C09095=1097.817,317.270,-83.466,178.547,18.904,152.358
C09096=1097.823,317.519,-83.498,178.550,18.907,152.358
C09097=1097.828,317.767,-83.529,178.553,18.909,152.358
C09098=1097.834,318.015,-83.561,178.556,18.912,152.358
C09099=1097.840,318.263,-83.593,178.560,18.915,152.358
C09100=1097.846,318.511,-83.625,178.563,18.918,152.358
C09101=1097.851,318.758,-83.657,178.566,18.920,152.359
C09102=1097.856,319.007,-83.689,178.569,18.923,152.359
C09103=1097.862,319.254,-83.721,178.572,18.926,152.359
C09104=1097.868,319.503,-83.753,178.575,18.928,152.359
C09105=1097.873,319.750,-83.785,178.578,18.931,152.359
C09106=1097.879,319.998,-83.817,178.583,18.934,152.359
C09107=1097.884,320.246,-83.848,178.586,18.937,152.359
C09108=1097.890,320.494,-83.880,178.589,18.939,152.359
C09109=1097.896,320.741,-83.912,178.592,18.942,152.359
C09110=1097.902,320.990,-83.944,178.595,18.945,152.359
C09111=1097.906,321.238,-83.976,178.598,18.948,152.359
C09112=1097.912,321.486,-84.008,178.601,18.951,152.359
C09113=1097.918,321.733,-84.040,178.604,18.954,152.359
C09114=1097.924,321.981,-84.072,178.607,18.956,152.359
C09115=1097.930,322.229,-84.105,178.611,18.959,152.359
C09116=1097.935,322.477,-84.136,178.614,18.961,152.360
C09117=1097.941,322.725,-84.169,178.618,18.965,152.360
C09118=1097.946,322.973,-84.201,178.621,18.967,152.360
C09119=1097.952,323.221,-84.233,178.624,18.970,152.360
C09120=1097.958,323.468,-84.266,178.627,18.973,152.360
C09121=1097.964,323.716,-84.297,178.630,18.975,152.360
C09122=1097.970,323.964,-84.329,178.633,18.979,152.360
C09123=1097.975,324.213,-84.362,178.637,18.981,152.360
C09124=1097.981,324.460,-84.394,178.640,18.984,152.360
C09125=1097.987,324.708,-84.426,178.643,18.987,152.360
C09126=1097.993,324.956,-84.458,178.646,18.990,152.360
C09127=1097.998,325.203,-84.491,178.649,18.993,152.360
C09128=1098.004,325.451,-84.523,178.652,18.996,152.361
C09129=1098.010,325.700,-84.555,178.655,18.998,152.361
C09130=1098.015,325.947,-84.588,178.658,19.001,152.361
C09131=1098.021,326.195,-84.620,178.661,19.004,152.361
C09132=1098.027,326.443,-84.652,178.665,19.007,152.361
C09133=1098.032,326.690,-84.685,178.668,19.010,152.361
C09134=1098.038,326.938,-84.717,178.671,19.013,152.361
C09135=1098.044,327.186,-84.750,178.674,19.016,152.361
C09136=1098.050,327.434,-84.782,178.678,19.019,152.361
C09137=1098.055,327.681,-84.814,178.681,19.022,152.362
C09138=1098.061,327.930,-84.847,178.684,19.024,152.362
C09139=1098.067,328.177,-84.880,178.687,19.027,152.362
C09140=1098.073,328.426,-84.912,178.691,19.030,152.362
C09141=1098.078,328.673,-84.945,178.694,19.033,152.362
C09142=1098.084,328.921,-84.977,178.697,19.036,152.362
C09143=1098.090,329.169,-85.010,178.700,19.039,152.362
C09144=1098.099,329.550,-85.060,178.705,19.044,152.362
C09145=1098.108,329.930,-85.109,178.710,19.047,152.362
C09146=1098.116,330.311,-85.160,178.715,19.052,152.363
C09147=1098.126,330.692,-85.210,178.720,19.057,152.363
C09148=1098.132,330.940,-85.242,178.723,19.060,152.363
C09149=1098.137,331.188,-85.276,178.726,19.063,152.363
C09150=1098.144,331.435,-85.309,178.729,19.066,152.363
C09151=1098.148,331.683,-85.341,178.733,19.069,152.363
C09152=1098.155,331.931,-85.374,178.735,19.072,152.364
C09153=1098.160,332.179,-85.407,178.738,19.075,152.364
C09154=1098.166,332.427,-85.439,178.742,19.078,152.364
C09155=1098.172,332.675,-85.472,178.745,19.081,152.364
C09156=1098.178,332.922,-85.505,178.748,19.084,152.364
C09157=1098.183,333.170,-85.538,178.751,19.087,152.364
C09158=1098.188,333.418,-85.571,178.755,19.090,152.364
C09159=1098.194,333.666,-85.603,178.757,19.094,152.365
C09160=1098.200,333.914,-85.637,178.760,19.096,152.365
C09161=1098.206,334.162,-85.670,178.764,19.100,152.365
C09162=1098.212,334.409,-85.703,178.767,19.103,152.365
C09163=1098.217,334.656,-85.736,178.770,19.106,152.365
C09164=1098.223,334.904,-85.768,178.773,19.110,152.366
C09165=1098.229,335.152,-85.802,178.776,19.112,152.366
C09166=1098.234,335.400,-85.835,178.779,19.115,152.366
C09167=1098.240,335.648,-85.868,178.783,19.119,152.366
C09168=1098.246,335.895,-85.901,178.786,19.122,152.366
C09169=1098.252,336.143,-85.935,178.789,19.125,152.367
C09170=1098.257,336.391,-85.968,178.792,19.129,152.367
C09171=1098.263,336.639,-86.001,178.795,19.131,152.367
C09172=1098.269,336.887,-86.034,178.798,19.135,152.367
C09173=1098.274,337.134,-86.067,178.802,19.138,152.367
C09174=1098.280,337.382,-86.100,178.805,19.141,152.367
C09175=1098.286,337.629,-86.133,178.808,19.145,152.368
C09176=1098.291,337.877,-86.166,178.811,19.148,152.368
C09177=1098.297,338.125,-86.200,178.814,19.151,152.368
C09178=1098.303,338.373,-86.232,178.818,19.154,152.368
C09179=1098.309,338.621,-86.266,178.820,19.157,152.368
C09180=1098.314,338.868,-86.299,178.823,19.161,152.369
C09181=1098.320,339.116,-86.333,178.827,19.164,152.369
C09182=1098.326,339.364,-86.366,178.830,19.167,152.369
C09183=1098.331,339.612,-86.400,178.833,19.171,152.369
C09184=1098.337,339.859,-86.433,178.836,19.174,152.370
C09185=1098.342,340.107,-86.467,178.839,19.177,152.370
C09186=1098.349,340.354,-86.500,178.842,19.181,152.370
C09187=1098.355,340.602,-86.533,178.845,19.184,152.370
C09188=1098.360,340.850,-86.567,178.849,19.188,152.371
C09189=1098.366,341.098,-86.600,178.851,19.191,152.371
C09190=1098.372,341.345,-86.634,178.854,19.194,152.371
C09191=1098.377,341.593,-86.667,178.858,19.198,152.371
C09192=1098.383,341.841,-86.701,178.861,19.201,152.372
C09193=1098.389,342.088,-86.735,178.864,19.205,152.372
C09194=1098.394,342.336,-86.768,178.867,19.208,152.372
C09195=1098.400,342.584,-86.802,178.870,19.211,152.372
C09196=1098.409,342.959,-86.852,178.875,19.216,152.373
C09197=1098.417,343.333,-86.903,178.880,19.222,152.373
C09198=1098.426,343.709,-86.955,178.885,19.227,152.373
C09199=1098.434,344.082,-87.006,178.889,19.232,152.374
C09200=1098.440,344.330,-87.039,178.892,19.236,152.374
C09201=1098.446,344.578,-87.074,178.895,19.239,152.374
C09202=1098.452,344.826,-87.107,178.899,19.243,152.375
C09203=1098.458,345.073,-87.141,178.901,19.246,152.375
C09204=1098.463,345.321,-87.174,178.905,19.250,152.375
C09205=1098.469,345.569,-87.208,178.908,19.253,152.376
C09206=1098.475,345.816,-87.242,178.911,19.257,152.376
C09207=1098.481,346.064,-87.276,178.914,19.260,152.376
C09208=1098.486,346.311,-87.310,178.916,19.263,152.376
C09209=1098.491,346.559,-87.344,178.920,19.267,152.377
C09210=1098.497,346.807,-87.378,178.923,19.271,152.377
C09211=1098.503,347.055,-87.412,178.926,19.274,152.377
C09212=1098.509,347.302,-87.446,178.929,19.278,152.378
C09213=1098.515,347.550,-87.480,178.932,19.282,152.378
C09214=1098.520,347.797,-87.514,178.935,19.285,152.378
C09215=1098.526,348.045,-87.548,178.939,19.289,152.379
C09216=1098.532,348.292,-87.582,178.941,19.292,152.379
C09217=1098.537,348.540,-87.616,178.945,19.296,152.379
C09218=1098.544,348.788,-87.650,178.947,19.300,152.380
C09219=1098.549,349.036,-87.684,178.951,19.303,152.380
C09220=1098.555,349.283,-87.718,178.953,19.307,152.380
C09221=1098.560,349.531,-87.752,178.957,19.311,152.380
C09222=1098.566,349.778,-87.787,178.960,19.315,152.381
C09223=1098.571,350.025,-87.821,178.963,19.318,152.381
C09224=1098.578,350.273,-87.855,178.966,19.322,152.381
C09225=1098.583,350.521,-87.889,178.969,19.326,152.382
C09226=1098.589,350.769,-87.923,178.972,19.330,152.382
C09227=1098.594,351.016,-87.957,178.975,19.333,152.383
C09228=1098.600,351.263,-87.991,178.979,19.337,152.383
C09229=1098.606,351.512,-88.027,178.981,19.340,152.383
C09230=1098.612,351.759,-88.061,178.985,19.344,152.384
C09231=1098.618,352.006,-88.095,178.987,19.348,152.384
C09232=1098.623,352.254,-88.129,178.991,19.352,152.384
C09233=1098.629,352.502,-88.164,178.993,19.355,152.385
C09234=1098.635,352.749,-88.198,178.997,19.359,152.385
C09235=1098.640,352.997,-88.232,179.000,19.363,152.385
C09236=1098.647,353.245,-88.267,179.003,19.367,152.386
C09237=1098.652,353.492,-88.301,179.006,19.371,152.386
C09238=1098.658,353.739,-88.336,179.009,19.374,152.387
C09239=1098.663,353.987,-88.371,179.012,19.379,152.387
C09240=1098.670,354.235,-88.405,179.014,19.382,152.387
C09241=1098.675,354.482,-88.440,179.018,19.386,152.388
C09242=1098.681,354.729,-88.474,179.021,19.390,152.388
C09243=1098.686,354.977,-88.509,179.024,19.394,152.388
C09244=1098.692,355.225,-88.543,179.027,19.398,152.389
C09245=1098.698,355.472,-88.578,179.030,19.402,152.389
C09246=1098.703,355.719,-88.612,179.033,19.406,152.390
C09247=1098.709,355.968,-88.647,179.036,19.410,152.390
C09248=1098.717,356.344,-88.700,179.041,19.416,152.391
C09249=1098.726,356.721,-88.753,179.045,19.422,152.391
C09250=1098.735,357.098,-88.806,179.050,19.428,152.392
C09251=1098.744,357.476,-88.859,179.055,19.434,152.393
C09252=1098.750,357.723,-88.894,179.057,19.438,152.393
C09253=1098.756,357.970,-88.929,179.060,19.442,152.393
C09254=1098.761,358.218,-88.964,179.064,19.446,152.394
C09255=1098.767,358.465,-88.998,179.066,19.450,152.394
C09256=1098.773,358.712,-89.033,179.069,19.454,152.395
C09257=1098.778,358.961,-89.068,179.073,19.458,152.395
C09258=1098.785,359.207,-89.103,179.075,19.462,152.396
C09259=1098.790,359.456,-89.138,179.079,19.466,152.396
C09260=1098.796,359.703,-89.173,179.082,19.471,152.397
C09261=1098.802,359.950,-89.207,179.084,19.475,152.397
C09262=1098.808,360.198,-89.243,179.088,19.479,152.397
C09263=1098.813,360.445,-89.278,179.091,19.483,152.398
C09264=1098.820,360.693,-89.313,179.093,19.487,152.398
C09265=1098.825,360.940,-89.347,179.096,19.491,152.399
C09266=1098.830,361.187,-89.383,179.100,19.495,152.399
C09267=1098.836,361.435,-89.418,179.102,19.499,152.400
C09268=1098.841,361.682,-89.453,179.105,19.504,152.400
C09269=1098.848,361.930,-89.488,179.109,19.508,152.401
C09270=1098.853,362.177,-89.524,179.111,19.512,152.401
C09271=1098.859,362.425,-89.559,179.114,19.517,152.402
C09272=1098.865,362.672,-89.594,179.117,19.521,152.402
C09273=1098.871,362.919,-89.629,179.120,19.525,152.403
C09274=1098.876,363.167,-89.664,179.123,19.529,152.403
C09275=1098.882,363.414,-89.699,179.126,19.534,152.404
C09276=1098.888,363.662,-89.735,179.129,19.538,152.404
C09277=1098.893,363.909,-89.770,179.132,19.542,152.405
C09278=1098.899,364.157,-89.805,179.135,19.546,152.405
C09279=1098.905,364.404,-89.841,179.138,19.551,152.406
C09280=1098.911,364.651,-89.876,179.140,19.555,152.406
C09281=1098.917,364.898,-89.911,179.144,19.559,152.407
C09282=1098.923,365.146,-89.947,179.147,19.563,152.407
C09283=1098.928,365.393,-89.982,179.150,19.568,152.408
C09284=1098.934,365.640,-90.018,179.152,19.572,152.408
C09285=1098.939,365.888,-90.053,179.156,19.576,152.409
C09286=1098.945,366.136,-90.088,179.159,19.581,152.410
C09287=1098.951,366.383,-90.124,179.162,19.586,152.410
C09288=1098.957,366.630,-90.159,179.164,19.590,152.411
C09289=1098.962,366.877,-90.195,179.167,19.594,152.411
C09290=1098.968,367.125,-90.230,179.170,19.599,152.412
C09291=1098.974,367.372,-90.266,179.173,19.604,152.412
C09292=1098.980,367.620,-90.302,179.175,19.608,152.413
C09293=1098.985,367.867,-90.337,179.179,19.612,152.414
C09294=1098.991,368.114,-90.373,179.182,19.617,152.414
C09295=1098.997,368.362,-90.408,179.185,19.621,152.415
C09296=1099.002,368.609,-90.444,179.188,19.626,152.415
C09297=1099.008,368.856,-90.481,179.190,19.630,152.416
C09298=1099.014,369.103,-90.516,179.193,19.635,152.416
C09299=1099.020,369.351,-90.552,179.196,19.640,152.417
C09300=1099.028,369.743,-90.608,179.201,19.647,152.418
C09301=1099.038,370.134,-90.665,179.205,19.654,152.419
C09302=1099.047,370.527,-90.722,179.210,19.662,152.420
C09303=1099.056,370.919,-90.778,179.214,19.669,152.421
C09304=1099.062,371.166,-90.815,179.217,19.674,152.422
C09305=1099.068,371.413,-90.850,179.220,19.678,152.422
C09306=1099.073,371.661,-90.886,179.223,19.683,152.423
C09307=1099.079,371.909,-90.922,179.226,19.688,152.423
C09308=1099.085,372.155,-90.958,179.229,19.693,152.424
C09309=1099.091,372.403,-90.994,179.231,19.697,152.425
C09310=1099.097,372.650,-91.030,179.234,19.702,152.425
C09311=1099.102,372.897,-91.066,179.237,19.706,152.426
C09312=1099.108,373.145,-91.102,179.240,19.711,152.427
C09313=1099.114,373.392,-91.138,179.243,19.716,152.427
C09314=1099.120,373.640,-91.174,179.246,19.721,152.428
C09315=1099.126,373.886,-91.210,179.249,19.726,152.429
C09316=1099.131,374.134,-91.247,179.251,19.730,152.429
C09317=1099.138,374.381,-91.283,179.254,19.735,152.430
C09318=1099.143,374.628,-91.318,179.257,19.740,152.431
C09319=1099.149,374.876,-91.355,179.260,19.745,152.431
C09320=1099.155,375.123,-91.391,179.263,19.750,152.432
C09321=1099.160,375.370,-91.428,179.266,19.755,152.433
C09322=1099.166,375.618,-91.464,179.269,19.760,152.433
C09323=1099.172,375.865,-91.500,179.272,19.765,152.434
C09324=1099.177,376.112,-91.536,179.275,19.770,152.435
C09325=1099.183,376.359,-91.572,179.277,19.775,152.436
C09326=1099.189,376.606,-91.609,179.280,19.779,152.436
C09327=1099.195,376.854,-91.645,179.283,19.784,152.437
C09328=1099.200,377.101,-91.682,179.286,19.789,152.438
C09329=1099.206,377.348,-91.718,179.288,19.795,152.439
C09330=1099.212,377.595,-91.754,179.291,19.800,152.439
C09331=1099.218,377.843,-91.791,179.294,19.805,152.440
C09332=1099.223,378.089,-91.827,179.297,19.810,152.441
C09333=1099.229,378.336,-91.864,179.300,19.815,152.441
C09334=1099.235,378.584,-91.900,179.302,19.820,152.442
C09335=1099.241,378.831,-91.937,179.305,19.825,152.443
C09336=1099.246,379.078,-91.973,179.308,19.831,152.444
C09337=1099.252,379.325,-92.010,179.311,19.835,152.444
C09338=1099.258,379.572,-92.047,179.314,19.841,152.445
C09339=1099.264,379.820,-92.083,179.317,19.846,152.446
C09340=1099.269,380.068,-92.120,179.319,19.851,152.447
C09341=1099.275,380.314,-92.156,179.322,19.856,152.448
C09342=1099.281,380.561,-92.193,179.325,19.861,152.448
C09343=1099.287,380.808,-92.229,179.328,19.867,152.449
C09344=1099.292,381.056,-92.267,179.331,19.872,152.450
C09345=1099.299,381.303,-92.303,179.333,19.877,152.451
C09346=1099.304,381.550,-92.340,179.336,19.882,152.452
C09347=1099.311,381.797,-92.376,179.339,19.887,152.452
C09348=1099.316,382.044,-92.413,179.342,19.893,152.453
C09349=1099.321,382.291,-92.450,179.344,19.898,152.454
C09350=1099.328,382.538,-92.487,179.347,19.903,152.455
C09351=1099.333,382.786,-92.524,179.350,19.909,152.456
C09352=1099.339,382.995,-92.555,179.352,19.913,152.456
C09353=1099.343,383.204,-92.586,179.354,19.917,152.457
C09354=1099.348,383.415,-92.617,179.356,19.922,152.458
C09355=1099.353,383.624,-92.649,179.359,19.927,152.458
C09356=1099.358,383.834,-92.680,179.361,19.931,152.459
C09357=1099.363,384.042,-92.712,179.363,19.936,152.460
C09358=1099.368,384.252,-92.743,179.366,19.941,152.461
C09359=1099.372,384.463,-92.774,179.368,19.946,152.461
C09360=1099.378,384.709,-92.811,179.371,19.951,152.462
C09361=1099.384,384.956,-92.848,179.374,19.956,152.463
C09362=1099.389,385.203,-92.885,179.376,19.962,152.464
C09363=1099.395,385.451,-92.922,179.379,19.967,152.465
C09364=1099.401,385.697,-92.960,179.381,19.973,152.466
C09365=1099.407,385.945,-92.997,179.384,19.978,152.467
C09366=1099.413,386.192,-93.034,179.387,19.984,152.467
C09367=1099.419,386.439,-93.071,179.390,19.990,152.468
C09368=1099.424,386.686,-93.108,179.393,19.995,152.469
C09369=1099.430,386.933,-93.145,179.395,20.001,152.470
C09370=1099.436,387.180,-93.183,179.398,20.007,152.471
C09371=1099.441,387.427,-93.220,179.400,20.012,152.472
C09372=1099.447,387.675,-93.257,179.403,20.018,152.473
C09373=1099.454,387.921,-93.294,179.406,20.023,152.474
C09374=1099.459,388.169,-93.331,179.408,20.029,152.475
C09375=1099.465,388.415,-93.369,179.412,20.035,152.476
C09376=1099.471,388.663,-93.406,179.414,20.041,152.477
C09377=1099.477,388.909,-93.444,179.417,20.047,152.478
C09378=1099.482,389.157,-93.481,179.419,20.052,152.479
C09379=1099.488,389.403,-93.519,179.422,20.058,152.479
C09380=1099.494,389.651,-93.556,179.425,20.063,152.480
C09381=1099.500,389.898,-93.594,179.428,20.070,152.481
C09382=1099.506,390.144,-93.631,179.430,20.075,152.482
C09383=1099.511,390.392,-93.668,179.433,20.081,152.483
C09384=1099.517,390.638,-93.706,179.435,20.087,152.484
C09385=1099.523,390.886,-93.743,179.438,20.093,152.485
C09386=1099.529,391.133,-93.781,179.440,20.098,152.486
C09387=1099.535,391.379,-93.819,179.444,20.105,152.487
C09388=1099.540,391.627,-93.856,179.446,20.110,152.488
C09389=1099.546,391.873,-93.894,179.449,20.116,152.489
C09390=1099.553,392.121,-93.932,179.451,20.122,152.490
C09391=1099.558,392.368,-93.969,179.454,20.128,152.491
C09392=1099.564,392.615,-94.006,179.457,20.134,152.492
C09393=1099.570,392.862,-94.044,179.459,20.141,152.493
C09394=1099.576,393.108,-94.082,179.462,20.146,152.494
C09395=1099.582,393.355,-94.120,179.464,20.152,152.495
C09396=1099.587,393.603,-94.157,179.467,20.159,152.496
C09397=1099.593,393.850,-94.195,179.470,20.165,152.498
C09398=1099.599,394.097,-94.233,179.472,20.171,152.499
C09399=1099.605,394.344,-94.271,179.475,20.177,152.500
C09400=1099.611,394.591,-94.309,179.478,20.184,152.501
C09401=1099.616,394.838,-94.347,179.480,20.189,152.502
C09402=1099.622,395.084,-94.385,179.482,20.195,152.503
C09403=1099.628,395.332,-94.423,179.485,20.202,152.504
C09404=1099.634,395.579,-94.461,179.488,20.208,152.505
C09405=1099.639,395.826,-94.499,179.490,20.214,152.506
C09406=1099.645,396.072,-94.537,179.493,20.221,152.507
C09407=1099.651,396.319,-94.575,179.495,20.227,152.508
C09408=1099.656,396.536,-94.607,179.497,20.233,152.509
C09409=1099.661,396.752,-94.641,179.500,20.238,152.510
C09410=1099.666,396.967,-94.674,179.502,20.243,152.511
C09411=1099.672,397.183,-94.707,179.504,20.249,152.512
C09412=1099.677,397.399,-94.741,179.507,20.255,152.513
C09413=1099.681,397.615,-94.775,179.508,20.260,152.514
C09414=1099.687,397.831,-94.808,179.511,20.266,152.515
C09415=1099.691,398.046,-94.841,179.513,20.272,152.516
C09416=1099.698,398.294,-94.879,179.516,20.278,152.518
C09417=1099.703,398.541,-94.917,179.518,20.284,152.519
C09418=1099.709,398.787,-94.956,179.521,20.291,152.520
C09419=1099.715,399.035,-94.994,179.523,20.298,152.521
C09420=1099.721,399.281,-95.032,179.525,20.304,152.522
C09421=1099.727,399.528,-95.070,179.528,20.311,152.523
C09422=1099.733,399.776,-95.109,179.531,20.317,152.525
C09423=1099.739,400.022,-95.147,179.533,20.323,152.526
C09424=1099.744,400.269,-95.185,179.536,20.331,152.527
C09425=1099.750,400.517,-95.224,179.538,20.337,152.528
C09426=1099.756,400.763,-95.263,179.541,20.344,152.529
C09427=1099.761,401.010,-95.301,179.543,20.350,152.531
C09428=1099.768,401.257,-95.339,179.545,20.357,152.532
C09429=1099.773,401.504,-95.378,179.548,20.364,152.533
C09430=1099.779,401.751,-95.416,179.550,20.371,152.534
C09431=1099.785,401.998,-95.455,179.553,20.378,152.536
C09432=1099.790,402.245,-95.494,179.555,20.384,152.537
C09433=1099.797,402.492,-95.532,179.558,20.391,152.538
C09434=1099.802,402.739,-95.571,179.560,20.398,152.539
C09435=1099.808,402.985,-95.609,179.563,20.405,152.541
C09436=1099.814,403.233,-95.648,179.565,20.412,152.542
C09437=1099.819,403.480,-95.686,179.568,20.418,152.543
C09438=1099.826,403.726,-95.725,179.570,20.426,152.545
C09439=1099.831,403.973,-95.764,179.572,20.432,152.546
C09440=1099.837,404.221,-95.803,179.575,20.439,152.547
C09441=1099.843,404.467,-95.841,179.577,20.446,152.549
C09442=1099.849,404.714,-95.880,179.580,20.453,152.550
C09443=1099.855,404.961,-95.919,179.583,20.461,152.551
C09444=1099.861,405.208,-95.957,179.585,20.467,152.552
C09445=1099.867,405.455,-95.997,179.588,20.475,152.554
C09446=1099.872,405.701,-96.036,179.590,20.482,152.555
C09447=1099.878,405.949,-96.074,179.593,20.489,152.557
C09448=1099.884,406.195,-96.113,179.595,20.496,152.558
C09449=1099.890,406.442,-96.152,179.597,20.504,152.559
C09450=1099.896,406.689,-96.191,179.599,20.510,152.561
C09451=1099.902,406.936,-96.230,179.602,20.518,152.562
C09452=1099.907,407.183,-96.269,179.605,20.525,152.564
C09453=1099.913,407.430,-96.308,179.607,20.532,152.565
C09454=1099.919,407.676,-96.348,179.609,20.540,152.566
C09455=1099.925,407.924,-96.386,179.611,20.547,152.568
C09456=1099.931,408.170,-96.425,179.614,20.554,152.569
C09457=1099.937,408.417,-96.464,179.617,20.562,152.571
C09458=1099.942,408.664,-96.503,179.619,20.569,152.572
C09459=1099.948,408.911,-96.543,179.621,20.577,152.573
C09460=1099.954,409.157,-96.582,179.624,20.584,152.575
C09461=1099.960,409.405,-96.621,179.626,20.592,152.576
C09462=1099.966,409.652,-96.661,179.629,20.599,152.578
C09463=1099.971,409.898,-96.700,179.631,20.607,152.579
C09464=1099.976,410.114,-96.734,179.633,20.614,152.581
C09465=1099.981,410.331,-96.768,179.635,20.621,152.582
C09466=1099.986,410.546,-96.803,179.637,20.627,152.583
C09467=1099.992,410.763,-96.837,179.640,20.634,152.584
C09468=1099.996,410.978,-96.872,179.642,20.641,152.586
C09469=1100.001,411.194,-96.906,179.644,20.647,152.587
C09470=1100.007,411.410,-96.941,179.646,20.654,152.589
C09471=1100.012,411.626,-96.975,179.648,20.661,152.590
C09472=1100.018,411.873,-97.015,179.650,20.668,152.591
C09473=1100.023,412.119,-97.054,179.652,20.676,152.593
C09474=1100.029,412.366,-97.094,179.655,20.684,152.594
C09475=1100.035,412.614,-97.133,179.657,20.692,152.596
C09476=1100.041,412.860,-97.172,179.660,20.699,152.597
C09477=1100.047,413.107,-97.212,179.661,20.707,152.599
C09478=1100.053,413.354,-97.252,179.664,20.715,152.601
C09479=1100.059,413.600,-97.291,179.667,20.723,152.602
C09480=1100.065,413.847,-97.330,179.669,20.731,152.604
C09481=1100.071,414.094,-97.371,179.671,20.739,152.605
C09482=1100.076,414.340,-97.410,179.674,20.747,152.607
C09483=1100.082,414.588,-97.450,179.676,20.755,152.609
C09484=1100.088,414.834,-97.490,179.678,20.763,152.610
C09485=1100.094,415.081,-97.529,179.681,20.771,152.612
C09486=1100.100,415.327,-97.569,179.683,20.779,152.613
C09487=1100.106,415.574,-97.608,179.686,20.787,152.615
C09488=1100.112,415.821,-97.649,179.688,20.796,152.617
C09489=1100.118,416.068,-97.689,179.690,20.804,152.618
C09490=1100.124,416.314,-97.728,179.693,20.812,152.620
C09491=1100.130,416.561,-97.768,179.694,20.820,152.622
C09492=1100.136,416.808,-97.808,179.697,20.828,152.623
C09493=1100.142,417.055,-97.848,179.699,20.837,152.625
C09494=1100.147,417.301,-97.888,179.701,20.845,152.627
C09495=1100.153,417.548,-97.928,179.704,20.853,152.628
C09496=1100.159,417.795,-97.968,179.706,20.862,152.630
C09497=1100.166,418.041,-98.008,179.708,20.870,152.632
C09498=1100.170,418.288,-98.048,179.711,20.879,152.634
C09499=1100.177,418.535,-98.088,179.713,20.887,152.635
C09500=1100.182,418.781,-98.129,179.715,20.896,152.637
C09501=1100.188,419.029,-98.168,179.718,20.904,152.639
C09502=1100.195,419.275,-98.208,179.720,20.913,152.641
C09503=1100.200,419.521,-98.249,179.722,20.922,152.643
C09504=1100.206,419.768,-98.289,179.724,20.930,152.644
C09505=1100.212,420.015,-98.329,179.727,20.939,152.646
C09506=1100.218,420.262,-98.369,179.729,20.947,152.648
C09507=1100.223,420.509,-98.410,179.731,20.956,152.650
C09508=1100.230,420.755,-98.450,179.733,20.965,152.651
C09509=1100.236,421.002,-98.491,179.735,20.973,152.653
C09510=1100.241,421.248,-98.530,179.738,20.982,152.655
C09511=1100.247,421.494,-98.571,179.740,20.992,152.657
C09512=1100.253,421.741,-98.611,179.743,21.000,152.659
C09513=1100.259,421.988,-98.652,179.745,21.009,152.661
C09514=1100.265,422.234,-98.692,179.747,21.018,152.663
C09515=1100.271,422.481,-98.733,179.749,21.027,152.664
C09516=1100.277,422.728,-98.773,179.751,21.036,152.666
C09517=1100.283,422.975,-98.814,179.753,21.045,152.668
C09518=1100.289,423.221,-98.854,179.755,21.054,152.670
C09519=1100.295,423.468,-98.895,179.758,21.064,152.672
C09520=1100.300,423.690,-98.931,179.760,21.071,152.674
C09521=1100.305,423.913,-98.968,179.762,21.080,152.675
C09522=1100.310,424.136,-99.004,179.764,21.088,152.677
C09523=1100.316,424.358,-99.042,179.766,21.096,152.679
C09524=1100.322,424.581,-99.078,179.767,21.104,152.681
C09525=1100.327,424.804,-99.115,179.770,21.113,152.683
C09526=1100.332,425.027,-99.152,179.772,21.122,152.684
C09527=1100.337,425.250,-99.188,179.773,21.130,152.686
C09528=1100.343,425.496,-99.229,179.775,21.139,152.688
C09529=1100.349,425.743,-99.270,179.778,21.149,152.690
C09530=1100.354,425.989,-99.311,179.780,21.158,152.692
C09531=1100.361,426.236,-99.351,179.782,21.167,152.694
C09532=1100.367,426.482,-99.393,179.784,21.177,152.696
C09533=1100.372,426.729,-99.433,179.787,21.187,152.698
C09534=1100.378,426.975,-99.475,179.789,21.196,152.700
C09535=1100.384,427.222,-99.516,179.791,21.205,152.702
C09536=1100.390,427.468,-99.556,179.793,21.215,152.704
C09537=1100.396,427.715,-99.597,179.795,21.225,152.706
C09538=1100.402,427.961,-99.638,179.797,21.234,152.709
C09539=1100.408,428.208,-99.679,179.799,21.244,152.711
C09540=1100.414,428.454,-99.721,179.802,21.254,152.713
C09541=1100.421,428.701,-99.761,179.804,21.264,152.715
C09542=1100.427,428.947,-99.803,179.805,21.273,152.717
C09543=1100.432,429.194,-99.844,179.808,21.283,152.719
C09544=1100.438,429.440,-99.885,179.810,21.293,152.721
C09545=1100.444,429.687,-99.927,179.812,21.304,152.724
C09546=1100.450,429.933,-99.967,179.814,21.313,152.726
C09547=1100.456,430.180,-100.009,179.816,21.323,152.728
C09548=1100.462,430.426,-100.050,179.818,21.334,152.730
C09549=1100.467,430.673,-100.091,179.820,21.343,152.732
C09550=1100.473,430.919,-100.132,179.823,21.354,152.734
C09551=1100.479,431.165,-100.174,179.824,21.364,152.737
C09552=1100.485,431.411,-100.215,179.826,21.374,152.739
C09553=1100.492,431.658,-100.257,179.829,21.384,152.741
C09554=1100.498,431.905,-100.298,179.830,21.394,152.743
C09555=1100.503,432.151,-100.339,179.833,21.405,152.746
C09556=1100.509,432.397,-100.381,179.834,21.415,152.748
C09557=1100.515,432.644,-100.422,179.837,21.426,152.750
C09558=1100.521,432.890,-100.464,179.838,21.436,152.753
C09559=1100.527,433.136,-100.506,179.841,21.446,152.755
C09560=1100.533,433.383,-100.548,179.843,21.457,152.757
C09561=1100.539,433.629,-100.589,179.845,21.467,152.759
C09562=1100.545,433.876,-100.631,179.846,21.478,152.762
C09563=1100.551,434.122,-100.672,179.849,21.488,152.764
C09564=1100.556,434.368,-100.714,179.850,21.499,152.767
C09565=1100.562,434.615,-100.755,179.853,21.510,152.769
C09566=1100.569,434.861,-100.797,179.854,21.520,152.771
C09567=1100.575,435.108,-100.839,179.856,21.532,152.774
C09568=1100.580,435.354,-100.882,179.858,21.542,152.776
C09569=1100.586,435.600,-100.923,179.860,21.553,152.779
C09570=1100.592,435.846,-100.964,179.862,21.564,152.781
C09571=1100.599,436.093,-101.006,179.864,21.575,152.784
C09572=1100.604,436.339,-101.048,179.866,21.586,152.786
C09573=1100.610,436.585,-101.090,179.868,21.596,152.788
C09574=1100.616,436.831,-101.132,179.870,21.608,152.791
C09575=1100.622,437.078,-101.174,179.872,21.619,152.794
C09576=1100.630,437.434,-101.235,179.874,21.635,152.797
C09577=1100.639,437.789,-101.296,179.877,21.651,152.801
C09578=1100.648,438.146,-101.356,179.879,21.667,152.804
C09579=1100.656,438.502,-101.418,179.882,21.684,152.808
C09580=1100.663,438.748,-101.460,179.884,21.695,152.811
C09581=1100.669,438.995,-101.502,179.886,21.706,152.813
C09582=1100.674,439.241,-101.544,179.888,21.718,152.816
C09583=1100.681,439.487,-101.586,179.890,21.730,152.819
C09584=1100.687,439.733,-101.628,179.892,21.741,152.821
C09585=1100.692,439.980,-101.670,179.893,21.752,152.824
C09586=1100.699,440.226,-101.713,179.895,21.764,152.826
C09587=1100.705,440.472,-101.756,179.897,21.776,152.829
C09588=1100.711,440.718,-101.797,179.899,21.788,152.832
C09589=1100.717,440.965,-101.840,179.900,21.799,152.835
C09590=1100.723,441.210,-101.882,179.902,21.811,152.837
C09591=1100.729,441.457,-101.925,179.904,21.823,152.840
C09592=1100.734,441.703,-101.968,179.906,21.835,152.843
C09593=1100.740,441.949,-102.010,179.907,21.846,152.845
C09594=1100.747,442.195,-102.053,179.909,21.858,152.848
C09595=1100.753,442.441,-102.095,179.911,21.871,152.851
C09596=1100.758,442.687,-102.138,179.913,21.883,152.854
C09597=1100.764,442.934,-102.180,179.915,21.895,152.857
C09598=1100.770,443.180,-102.222,179.917,21.907,152.859
C09599=1100.777,443.426,-102.266,179.918,21.919,152.862
C09600=1100.782,443.672,-102.308,179.919,21.931,152.865
C09601=1100.789,443.918,-102.351,179.921,21.944,152.868
C09602=1100.794,444.164,-102.394,179.922,21.956,152.871
C09603=1100.801,444.411,-102.437,179.924,21.968,152.874
C09604=1100.806,444.657,-102.480,179.925,21.980,152.877
C09605=1100.813,444.903,-102.522,179.926,21.992,152.880
C09606=1100.818,445.149,-102.565,179.926,22.005,152.883
C09607=1100.825,445.396,-102.608,179.927,22.017,152.886
C09608=1100.830,445.641,-102.651,179.927,22.028,152.889
C09609=1100.837,445.888,-102.693,179.928,22.041,152.892
C09610=1100.843,446.133,-102.737,179.928,22.053,152.895
C09611=1100.849,446.380,-102.780,179.928,22.065,152.898
C09612=1100.854,446.626,-102.823,179.928,22.077,152.901
C09613=1100.861,446.872,-102.866,179.928,22.089,152.904
C09614=1100.866,447.118,-102.909,179.928,22.101,152.907
C09615=1100.872,447.365,-102.952,179.927,22.113,152.910
C09616=1100.879,447.611,-102.996,179.926,22.125,152.913
C09617=1100.884,447.856,-103.038,179.925,22.137,152.916
C09618=1100.890,448.103,-103.081,179.925,22.149,152.920
C09619=1100.896,448.349,-103.124,179.924,22.161,152.923
C09620=1100.903,448.595,-103.167,179.923,22.173,152.926
C09621=1100.909,448.841,-103.211,179.923,22.185,152.929
C09622=1100.915,449.087,-103.253,179.921,22.197,152.932
C09623=1100.921,449.333,-103.297,179.919,22.209,152.936
C09624=1100.926,449.579,-103.340,179.918,22.221,152.939
C09625=1100.933,449.826,-103.383,179.917,22.233,152.942
C09626=1100.938,450.071,-103.427,179.915,22.244,152.945
C09627=1100.945,450.317,-103.470,179.914,22.256,152.948
C09628=1100.547,450.310,-103.615,179.847,22.478,153.015
C09629=1100.541,450.064,-103.571,179.849,22.467,153.012
C09630=1100.534,449.818,-103.529,179.850,22.454,153.008
C09631=1100.528,449.571,-103.485,179.851,22.442,153.005
C09632=1100.522,449.326,-103.442,179.853,22.431,153.002
C09633=1100.516,449.080,-103.399,179.854,22.419,152.999
C09634=1100.510,448.834,-103.355,179.855,22.407,152.996
C09635=1100.504,448.588,-103.312,179.856,22.395,152.992
C09636=1100.498,448.341,-103.269,179.857,22.383,152.989
C09637=1100.492,448.096,-103.226,179.858,22.370,152.986
C09638=1100.486,447.849,-103.182,179.859,22.359,152.983
C09639=1100.480,447.603,-103.139,179.859,22.346,152.980
C09640=1100.474,447.357,-103.096,179.860,22.334,152.976
C09641=1100.468,447.111,-103.053,179.860,22.322,152.973
C09642=1100.462,446.865,-103.010,179.860,22.310,152.970
C09643=1100.456,446.618,-102.967,179.860,22.298,152.967
C09644=1100.450,446.372,-102.923,179.860,22.286,152.964
C09645=1100.444,446.126,-102.880,179.861,22.274,152.961
C09646=1100.437,445.880,-102.838,179.860,22.261,152.958
C09647=1100.432,445.634,-102.795,179.860,22.249,152.955
C09648=1100.426,445.388,-102.752,179.859,22.237,152.952
C09649=1100.420,445.142,-102.709,179.858,22.225,152.949
C09650=1100.414,444.896,-102.665,179.857,22.212,152.946
C09651=1100.407,444.650,-102.623,179.856,22.200,152.943
C09652=1100.401,444.404,-102.580,179.855,22.188,152.940
C09653=1100.395,444.157,-102.537,179.855,22.176,152.937
C09654=1100.390,443.911,-102.494,179.853,22.163,152.934
C09655=1100.383,443.665,-102.451,179.852,22.151,152.931
C09656=1100.377,443.419,-102.409,179.850,22.139,152.928
C09657=1100.372,443.173,-102.366,179.848,22.127,152.926
C09658=1100.366,442.926,-102.323,179.846,22.114,152.923
C09659=1100.359,442.681,-102.281,179.844,22.102,152.920
C09660=1100.353,442.434,-102.237,179.842,22.090,152.917
C09661=1100.348,442.188,-102.195,179.841,22.078,152.914
C09662=1100.341,441.942,-102.152,179.839,22.066,152.911
C09663=1100.336,441.696,-102.110,179.837,22.054,152.909
C09664=1100.329,441.450,-102.068,179.835,22.041,152.906
C09665=1100.323,441.203,-102.025,179.833,22.029,152.903
C09666=1100.318,440.958,-101.982,179.832,22.018,152.900
C09667=1100.311,440.711,-101.939,179.830,22.006,152.898
C09668=1100.306,440.465,-101.897,179.828,21.994,152.895
C09669=1100.299,440.219,-101.855,179.826,21.982,152.892
C09670=1100.293,439.973,-101.812,179.824,21.971,152.890
C09671=1100.287,439.726,-101.771,179.822,21.959,152.887
C09672=1100.280,439.480,-101.728,179.820,21.948,152.884
C09673=1100.275,439.234,-101.685,179.818,21.936,152.882
C09674=1100.269,438.988,-101.644,179.817,21.925,152.879
C09675=1100.263,438.741,-101.601,179.814,21.913,152.877
C09676=1100.257,438.495,-101.559,179.812,21.902,152.874
C09677=1100.248,438.146,-101.499,179.810,21.886,152.870
C09678=1100.240,437.797,-101.439,179.807,21.870,152.867
C09679=1100.231,437.449,-101.380,179.804,21.854,152.863
C09680=1100.223,437.100,-101.321,179.802,21.838,152.860
C09681=1100.217,436.853,-101.278,179.800,21.827,152.857
C09682=1100.210,436.607,-101.236,179.797,21.815,152.854
C09683=1100.205,436.361,-101.195,179.796,21.804,152.852
C09684=1100.199,436.115,-101.152,179.794,21.793,152.850
C09685=1100.192,435.868,-101.110,179.791,21.782,152.847
C09686=1100.187,435.622,-101.068,179.790,21.771,152.845
C09687=1100.181,435.376,-101.026,179.788,21.760,152.842
C09688=1100.175,435.130,-100.985,179.786,21.750,152.840
C09689=1100.168,434.883,-100.942,179.784,21.739,152.837
C09690=1100.163,434.637,-100.900,179.782,21.728,152.835
C09691=1100.157,434.391,-100.859,179.780,21.717,152.833
C09692=1100.151,434.144,-100.817,179.778,21.706,152.830
C09693=1100.145,433.898,-100.776,179.776,21.696,152.828
C09694=1100.140,433.651,-100.734,179.773,21.685,152.825
C09695=1100.134,433.405,-100.692,179.772,21.674,152.823
C09696=1100.128,433.158,-100.651,179.769,21.663,152.821
C09697=1100.122,432.912,-100.609,179.768,21.653,152.818
C09698=1100.116,432.666,-100.568,179.766,21.643,152.816
C09699=1100.110,432.420,-100.526,179.763,21.632,152.814
C09700=1100.103,432.173,-100.484,179.762,21.622,152.811
C09701=1100.097,431.927,-100.443,179.759,21.612,152.809
C09702=1100.091,431.681,-100.402,179.758,21.601,152.807
C09703=1100.085,431.434,-100.360,179.755,21.591,152.805
C09704=1100.080,431.188,-100.318,179.753,21.581,152.802
C09705=1100.074,430.942,-100.277,179.751,21.570,152.800
C09706=1100.069,430.695,-100.236,179.749,21.560,152.798
C09707=1100.062,430.448,-100.194,179.747,21.550,152.796
C09708=1100.056,430.202,-100.153,179.744,21.540,152.794
C09709=1100.050,429.956,-100.111,179.743,21.530,152.791
C09710=1100.045,429.709,-100.070,179.740,21.520,152.789
C09711=1100.039,429.462,-100.029,179.738,21.510,152.787
C09712=1100.033,429.216,-99.987,179.737,21.500,152.785
C09713=1100.027,428.970,-99.946,179.734,21.489,152.783
C09714=1100.020,428.724,-99.906,179.732,21.480,152.780
C09715=1100.014,428.477,-99.864,179.730,21.470,152.778
C09716=1100.009,428.231,-99.824,179.727,21.460,152.776
C09717=1100.002,427.984,-99.782,179.725,21.451,152.774
C09718=1099.997,427.737,-99.741,179.723,21.441,152.772
C09719=1099.991,427.491,-99.700,179.721,21.431,152.770
C09720=1099.984,427.245,-99.659,179.719,21.421,152.768
C09721=1099.978,426.998,-99.618,179.717,21.412,152.766
C09722=1099.973,426.751,-99.577,179.715,21.402,152.764
C09723=1099.967,426.505,-99.536,179.712,21.392,152.762
C09724=1099.961,426.258,-99.495,179.710,21.383,152.760
C09725=1099.954,426.012,-99.454,179.708,21.374,152.758
C09726=1099.949,425.765,-99.413,179.706,21.364,152.756
C09727=1099.943,425.518,-99.373,179.703,21.355,152.754
C09728=1099.937,425.272,-99.331,179.701,21.345,152.752
C09729=1099.932,425.050,-99.295,179.699,21.336,152.750
C09730=1099.927,424.826,-99.257,179.698,21.328,152.748
C09731=1099.921,424.603,-99.221,179.695,21.320,152.746
C09732=1099.915,424.380,-99.184,179.694,21.311,152.744
C09733=1099.911,424.157,-99.147,179.691,21.303,152.743
C09734=1099.905,423.934,-99.111,179.689,21.294,152.741
C09735=1099.900,423.711,-99.073,179.688,21.286,152.739
C09736=1099.894,423.488,-99.037,179.685,21.277,152.737
C09737=1099.889,423.241,-98.996,179.683,21.268,152.735
C09738=1099.882,422.994,-98.956,179.681,21.259,152.733
C09739=1099.877,422.747,-98.915,179.679,21.251,152.732
C09740=1099.871,422.501,-98.874,179.677,21.241,152.730
C09741=1099.865,422.255,-98.835,179.674,21.232,152.728
C09742=1099.860,422.008,-98.794,179.671,21.223,152.726
C09743=1099.853,421.761,-98.754,179.669,21.214,152.724
C09744=1099.847,421.515,-98.712,179.667,21.205,152.722
C09745=1099.841,421.268,-98.673,179.665,21.196,152.720
C09746=1099.835,421.021,-98.632,179.663,21.188,152.718
C09747=1099.829,420.775,-98.592,179.660,21.179,152.717
C09748=1099.823,420.528,-98.551,179.658,21.170,152.715
C09749=1099.817,420.281,-98.511,179.656,21.161,152.713
C09750=1099.811,420.035,-98.470,179.654,21.152,152.711
C09751=1099.806,419.789,-98.430,179.651,21.144,152.709
C09752=1099.800,419.542,-98.390,179.649,21.135,152.707
C09753=1099.794,419.295,-98.350,179.647,21.126,152.706
C09754=1099.788,419.048,-98.310,179.645,21.118,152.704
C09755=1099.782,418.801,-98.269,179.642,21.109,152.702
C09756=1099.776,418.555,-98.229,179.640,21.101,152.700
C09757=1099.770,418.309,-98.189,179.638,21.092,152.699
C09758=1099.764,418.062,-98.149,179.635,21.083,152.697
C09759=1099.759,417.815,-98.109,179.633,21.075,152.695
C09760=1099.752,417.568,-98.069,179.631,21.066,152.693
C09761=1099.746,417.321,-98.029,179.628,21.058,152.692
C09762=1099.741,417.075,-97.989,179.626,21.049,152.690
C09763=1099.735,416.829,-97.949,179.623,21.041,152.688
C09764=1099.730,416.581,-97.909,179.621,21.033,152.687
C09765=1099.723,416.335,-97.868,179.619,21.024,152.685
C09766=1099.718,416.088,-97.829,179.616,21.016,152.683
C09767=1099.711,415.842,-97.789,179.614,21.007,152.681
C09768=1099.705,415.595,-97.750,179.611,21.000,152.680
C09769=1099.700,415.348,-97.709,179.609,20.992,152.678
C09770=1099.694,415.101,-97.670,179.607,20.984,152.677
C09771=1099.688,414.855,-97.630,179.605,20.975,152.675
C09772=1099.682,414.608,-97.590,179.602,20.967,152.673
C09773=1099.675,414.361,-97.550,179.599,20.959,152.672
C09774=1099.669,414.114,-97.511,179.597,20.951,152.670
C09775=1099.665,413.867,-97.471,179.595,20.942,152.668
C09776=1099.658,413.621,-97.431,179.593,20.935,152.667
C09777=1099.652,413.374,-97.392,179.590,20.927,152.665
C09778=1099.647,413.127,-97.353,179.588,20.919,152.664
C09779=1099.640,412.881,-97.312,179.585,20.911,152.662
C09780=1099.634,412.633,-97.273,179.583,20.903,152.661
C09781=1099.628,412.386,-97.234,179.581,20.895,152.659
C09782=1099.623,412.140,-97.194,179.578,20.888,152.658
C09783=1099.616,411.893,-97.154,179.576,20.880,152.656
C09784=1099.611,411.647,-97.115,179.573,20.872,152.654
C09785=1099.606,411.430,-97.080,179.571,20.865,152.653
C09786=1099.601,411.214,-97.045,179.569,20.858,152.652
C09787=1099.596,410.998,-97.011,179.567,20.851,152.650
C09788=1099.591,410.781,-96.977,179.565,20.844,152.649
C09789=1099.585,410.565,-96.942,179.563,20.838,152.648
C09790=1099.581,410.349,-96.908,179.560,20.831,152.646
C09791=1099.575,410.133,-96.873,179.558,20.824,152.645
C09792=1099.571,409.916,-96.839,179.556,20.818,152.644
C09793=1099.564,409.670,-96.799,179.554,20.810,152.642
C09794=1099.558,409.423,-96.760,179.552,20.802,152.641
C09795=1099.553,409.176,-96.720,179.549,20.795,152.639
C09796=1099.547,408.929,-96.682,179.546,20.787,152.638
C09797=1099.541,408.682,-96.643,179.544,20.780,152.636
C09798=1099.535,408.435,-96.603,179.542,20.772,152.635
C09799=1099.530,408.189,-96.564,179.539,20.765,152.634
C09800=1099.524,407.941,-96.525,179.537,20.757,152.632
C09801=1099.518,407.695,-96.486,179.534,20.750,152.631
C09802=1099.512,407.448,-96.447,179.532,20.743,152.629
C09803=1099.506,407.202,-96.408,179.530,20.735,152.628
C09804=1099.500,406.955,-96.368,179.527,20.727,152.626
C09805=1099.495,406.708,-96.330,179.525,20.721,152.625
C09806=1099.489,406.460,-96.291,179.522,20.713,152.624
C09807=1099.483,406.214,-96.252,179.520,20.706,152.622
C09808=1099.476,405.967,-96.213,179.518,20.699,152.621
C09809=1099.471,405.720,-96.174,179.515,20.691,152.619
C09810=1099.465,405.473,-96.135,179.513,20.684,152.618
C09811=1099.460,405.227,-96.096,179.510,20.677,152.617
C09812=1099.453,404.979,-96.058,179.508,20.670,152.615
C09813=1099.448,404.733,-96.019,179.505,20.663,152.614
C09814=1099.442,404.486,-95.979,179.503,20.656,152.613
C09815=1099.437,404.238,-95.941,179.500,20.649,152.611
C09816=1099.430,403.992,-95.902,179.498,20.642,152.610
C09817=1099.424,403.745,-95.863,179.495,20.635,152.609
C09818=1099.418,403.497,-95.824,179.493,20.628,152.607
C09819=1099.412,403.251,-95.786,179.490,20.621,152.606
C09820=1099.406,403.004,-95.747,179.488,20.614,152.605
C09821=1099.401,402.757,-95.708,179.485,20.607,152.604
C09822=1099.395,402.510,-95.670,179.483,20.600,152.602
C09823=1099.389,402.263,-95.631,179.480,20.593,152.601
C09824=1099.383,402.017,-95.593,179.478,20.586,152.600
C09825=1099.377,401.769,-95.554,179.475,20.579,152.598
C09826=1099.372,401.522,-95.515,179.473,20.573,152.597
C09827=1099.366,401.276,-95.477,179.470,20.566,152.596
C09828=1099.360,401.028,-95.438,179.467,20.559,152.595
C09829=1099.354,400.782,-95.400,179.465,20.553,152.593
C09830=1099.348,400.534,-95.362,179.462,20.545,152.592
C09831=1099.342,400.288,-95.323,179.460,20.539,152.591
C09832=1099.337,400.041,-95.285,179.458,20.532,152.590
C09833=1099.332,399.794,-95.246,179.455,20.525,152.588
C09834=1099.325,399.547,-95.208,179.453,20.519,152.587
C09835=1099.319,399.300,-95.170,179.450,20.512,152.586
C09836=1099.313,399.052,-95.131,179.447,20.505,152.585
C09837=1099.307,398.806,-95.093,179.445,20.499,152.584
C09838=1099.302,398.559,-95.054,179.442,20.492,152.582
C09839=1099.296,398.312,-95.017,179.440,20.486,152.581
C09840=1099.290,398.065,-94.978,179.438,20.480,152.580
C09841=1099.285,397.849,-94.945,179.435,20.473,152.579
C09842=1099.280,397.633,-94.911,179.433,20.468,152.578
C09843=1099.275,397.416,-94.878,179.431,20.463,152.577
C09844=1099.270,397.200,-94.845,179.428,20.457,152.576
C09845=1099.265,396.985,-94.812,179.426,20.451,152.575
C09846=1099.259,396.768,-94.777,179.424,20.446,152.574
C09847=1099.254,396.552,-94.744,179.422,20.440,152.573
C09848=1099.249,396.336,-94.711,179.419,20.434,152.572
C09849=1099.244,396.089,-94.673,179.417,20.428,152.571
C09850=1099.238,395.842,-94.635,179.415,20.421,152.570
C09851=1099.232,395.596,-94.597,179.412,20.415,152.569
C09852=1099.226,395.348,-94.558,179.409,20.409,152.568
C09853=1099.220,395.101,-94.521,179.407,20.402,152.566
C09854=1099.215,394.854,-94.484,179.404,20.396,152.565
C09855=1099.209,394.607,-94.446,179.401,20.390,152.564
C09856=1099.203,394.360,-94.408,179.399,20.384,152.563
C09857=1099.197,394.112,-94.369,179.396,20.378,152.562
C09858=1099.191,393.866,-94.332,179.394,20.372,152.561
C09859=1099.185,393.619,-94.294,179.391,20.365,152.560
C09860=1099.179,393.372,-94.256,179.388,20.359,152.559
C09861=1099.173,393.125,-94.218,179.386,20.353,152.558
C09862=1099.169,392.878,-94.181,179.383,20.347,152.557
C09863=1099.163,392.631,-94.143,179.381,20.341,152.556
C09864=1099.156,392.384,-94.105,179.378,20.334,152.555
C09865=1099.150,392.137,-94.067,179.375,20.329,152.554
C09866=1099.145,391.889,-94.030,179.373,20.323,152.553
C09867=1099.139,391.643,-93.992,179.370,20.317,152.552
C09868=1099.133,391.396,-93.954,179.367,20.311,152.551
C09869=1099.127,391.149,-93.917,179.364,20.304,152.550
C09870=1099.121,390.902,-93.880,179.362,20.299,152.549
C09871=1099.115,390.654,-93.842,179.359,20.293,152.548
C09872=1099.109,390.408,-93.804,179.357,20.287,152.547
C09873=1099.103,390.160,-93.767,179.354,20.282,152.546
C09874=1099.097,389.914,-93.729,179.351,20.275,152.545
C09875=1099.092,389.666,-93.692,179.348,20.269,152.544
C09876=1099.086,389.420,-93.654,179.346,20.264,152.543
C09877=1099.080,389.173,-93.616,179.343,20.258,152.542
C09878=1099.074,388.925,-93.579,179.341,20.252,152.541
C09879=1099.068,388.679,-93.542,179.338,20.247,152.540
C09880=1099.063,388.431,-93.505,179.335,20.240,152.539
C09881=1099.057,388.185,-93.467,179.332,20.235,152.538
C09882=1099.051,387.937,-93.430,179.330,20.229,152.537
C09883=1099.045,387.691,-93.393,179.327,20.223,152.536
C09884=1099.039,387.443,-93.356,179.325,20.217,152.535
C09885=1099.033,387.197,-93.318,179.322,20.212,152.534
C09886=1099.028,386.949,-93.281,179.319,20.206,152.533
C09887=1099.022,386.702,-93.244,179.316,20.200,152.532
C09888=1099.016,386.455,-93.206,179.313,20.195,152.531
C09889=1099.011,386.208,-93.169,179.311,20.189,152.530
C09890=1099.004,385.961,-93.133,179.308,20.183,152.530
C09891=1098.998,385.714,-93.095,179.305,20.178,152.529
C09892=1098.993,385.467,-93.058,179.303,20.172,152.528
C09893=1098.987,385.219,-93.021,179.300,20.167,152.527
C09894=1098.982,384.973,-92.983,179.297,20.161,152.526
C09895=1098.976,384.726,-92.946,179.295,20.156,152.525
C09896=1098.970,384.479,-92.910,179.292,20.150,152.524
C09897=1098.965,384.268,-92.878,179.289,20.145,152.523
C09898=1098.960,384.059,-92.846,179.287,20.140,152.523
C09899=1098.956,383.849,-92.815,179.285,20.136,152.522
C09900=1098.951,383.639,-92.784,179.282,20.131,152.521
C09901=1098.946,383.429,-92.753,179.280,20.126,152.520
C09902=1098.941,383.219,-92.721,179.278,20.122,152.520
C09903=1098.936,383.009,-92.689,179.275,20.117,152.519
C09904=1098.931,382.800,-92.659,179.273,20.112,152.518
C09905=1098.926,382.553,-92.622,179.270,20.107,152.517
C09906=1098.919,382.306,-92.585,179.268,20.102,152.517
C09907=1098.914,382.059,-92.548,179.265,20.096,152.516
C09908=1098.907,381.812,-92.511,179.262,20.091,152.515
C09909=1098.902,381.564,-92.474,179.259,20.086,152.514
C09910=1098.896,381.317,-92.437,179.256,20.080,152.513
C09911=1098.890,381.070,-92.401,179.254,20.075,152.513
C09912=1098.885,380.823,-92.364,179.251,20.070,152.512
C09913=1098.878,380.576,-92.327,179.248,20.065,152.511
C09914=1098.873,380.328,-92.291,179.245,20.059,152.510
C09915=1098.867,380.081,-92.255,179.243,20.054,152.509
C09916=1098.861,379.834,-92.218,179.240,20.049,152.509
C09917=1098.856,379.587,-92.181,179.237,20.044,152.508
C09918=1098.849,379.339,-92.144,179.234,20.038,152.507
C09919=1098.844,379.093,-92.107,179.231,20.034,152.506
C09920=1098.838,378.846,-92.071,179.228,20.028,152.505
C09921=1098.832,378.598,-92.034,179.226,20.023,152.505
C09922=1098.826,378.351,-91.998,179.223,20.018,152.504
C09923=1098.821,378.104,-91.962,179.220,20.013,152.503
C09924=1098.815,377.857,-91.925,179.217,20.008,152.502
C09925=1098.809,377.610,-91.888,179.214,20.002,152.502
C09926=1098.803,377.362,-91.852,179.212,19.998,152.501
C09927=1098.798,377.115,-91.816,179.209,19.993,152.500
C09928=1098.792,376.868,-91.779,179.206,19.988,152.499
C09929=1098.786,376.621,-91.744,179.204,19.982,152.499
C09930=1098.780,376.373,-91.706,179.201,19.977,152.498
C09931=1098.775,376.127,-91.670,179.198,19.972,152.497
C09932=1098.769,375.879,-91.634,179.195,19.967,152.496
C09933=1098.763,375.632,-91.598,179.192,19.962,152.496
C09934=1098.757,375.384,-91.561,179.189,19.957,152.495
C09935=1098.752,375.137,-91.525,179.186,19.952,152.494
C09936=1098.746,374.890,-91.489,179.183,19.947,152.494
C09937=1098.740,374.642,-91.452,179.180,19.942,152.493
C09938=1098.735,374.396,-91.416,179.178,19.938,152.492
C09939=1098.729,374.148,-91.380,179.175,19.933,152.492
C09940=1098.723,373.901,-91.344,179.172,19.928,152.491
C09941=1098.717,373.654,-91.308,179.169,19.923,152.490
C09942=1098.711,373.407,-91.272,179.166,19.918,152.490
C09943=1098.705,373.159,-91.236,179.163,19.913,152.489
C09944=1098.700,372.913,-91.199,179.160,19.908,152.488
C09945=1098.694,372.665,-91.164,179.157,19.903,152.487
C09946=1098.688,372.417,-91.128,179.155,19.899,152.487
C09947=1098.682,372.170,-91.091,179.152,19.894,152.486
C09948=1098.676,371.923,-91.056,179.149,19.890,152.486
C09949=1098.671,371.675,-91.020,179.146,19.885,152.485
C09950=1098.665,371.428,-90.983,179.143,19.880,152.484
C09951=1098.659,371.181,-90.948,179.140,19.875,152.484
C09952=1098.653,370.934,-90.912,179.138,19.871,152.483
C09953=1098.644,370.541,-90.855,179.133,19.863,152.482
C09954=1098.635,370.149,-90.798,179.128,19.856,152.481
C09955=1098.626,369.756,-90.741,179.124,19.848,152.480
C09956=1098.616,369.364,-90.685,179.119,19.841,152.479
C09957=1098.611,369.117,-90.649,179.116,19.836,152.478
C09958=1098.605,368.869,-90.613,179.113,19.831,152.478
C09959=1098.600,368.621,-90.577,179.111,19.827,152.477
C09960=1098.594,368.374,-90.542,179.108,19.822,152.477
C09961=1098.588,368.126,-90.506,179.105,19.818,152.476
C09962=1098.582,367.880,-90.470,179.102,19.813,152.475
C09963=1098.576,367.632,-90.434,179.099,19.808,152.475
C09964=1098.571,367.385,-90.399,179.096,19.804,152.474
C09965=1098.565,367.138,-90.363,179.093,19.800,152.474
C09966=1098.560,366.891,-90.328,179.090,19.795,152.473
C09967=1098.554,366.643,-90.292,179.087,19.790,152.472
C09968=1098.548,366.396,-90.257,179.085,19.786,152.472
C09969=1098.542,366.148,-90.221,179.082,19.782,152.471
C09970=1098.537,365.901,-90.186,179.079,19.777,152.471
C09971=1098.531,365.653,-90.151,179.076,19.772,152.470
C09972=1098.526,365.406,-90.115,179.072,19.768,152.470
C09973=1098.519,365.158,-90.080,179.070,19.764,152.469
C09974=1098.513,364.911,-90.044,179.067,19.759,152.468
C09975=1098.508,364.664,-90.008,179.064,19.755,152.468
C09976=1098.502,364.416,-89.973,179.061,19.751,152.467
C09977=1098.497,364.169,-89.937,179.058,19.746,152.467
C09978=1098.490,363.921,-89.903,179.055,19.742,152.466
C09979=1098.485,363.674,-89.868,179.052,19.737,152.466
C09980=1098.479,363.426,-89.832,179.049,19.733,152.465
C09981=1098.473,363.180,-89.796,179.046,19.729,152.465
C09982=1098.468,362.932,-89.762,179.043,19.724,152.464
C09983=1098.462,362.684,-89.726,179.040,19.720,152.464
C09984=1098.456,362.438,-89.691,179.037,19.716,152.463
C09985=1098.450,362.190,-89.656,179.034,19.712,152.463
C09986=1098.445,361.942,-89.621,179.031,19.707,152.462
C09987=1098.439,361.695,-89.585,179.029,19.703,152.462
C09988=1098.433,361.448,-89.550,179.025,19.699,152.461
C09989=1098.427,361.200,-89.515,179.022,19.695,152.461
C09990=1098.421,360.953,-89.480,179.020,19.691,152.460
C09991=1098.416,360.705,-89.445,179.017,19.686,152.460
C09992=1098.410,360.457,-89.410,179.013,19.682,152.459
C09993=1098.404,360.211,-89.375,179.011,19.678,152.459
C09994=1098.398,359.962,-89.340,179.008,19.674,152.458
C09995=1098.393,359.715,-89.305,179.004,19.670,152.458
C09996=1098.386,359.468,-89.270,179.002,19.666,152.457
//INST
///DATE 2021/06/17 10:53
///ATTR SC,RW,RJ
////FRAME ROBOT
///GROUP1 RB1
NOP
MOVL C00000 V=800.0 PL=0
MOVL C00001 V=800.0 PL=0
MOVL C00002 V=800.0 PL=0
MOVL C00003 V=800.0 PL=0
MOVL C00004 V=800.0 PL=0
MOVL C00005 V=800.0 PL=0
MOVL C00006 V=800.0 PL=0
MOVL C00007 V=800.0 PL=0
MOVL C00008 V=800.0 PL=0
MOVL C00009 V=800.0 PL=0
MOVL C00010 V=800.0 PL=0
MOVL C00011 V=800.0 PL=0
MOVL C00012 V=800.0 PL=0
MOVL C00013 V=800.0 PL=0
MOVL C00014 V=800.0 PL=0
MOVL C00015 V=800.0 PL=0
MOVL C00016 V=800.0 PL=0
MOVL C00017 V=800.0 PL=0
MOVL C00018 V=800.0 PL=0
MOVL C00019 V=800.0 PL=0
MOVL C00020 V=800.0 PL=0
MOVL C00021 V=800.0 PL=0
MOVL C00022 V=800.0 PL=0
MOVL C00023 V=800.0 PL=0
MOVL C00024 V=800.0 PL=0
MOVL C00025 V=800.0 PL=0
MOVL C00026 V=800.0 PL=0
MOVL C00027 V=800.0 PL=0
MOVL C00028 V=800.0 PL=0
MOVL C00029 V=800.0 PL=0
MOVL C00030 V=800.0 PL=0
MOVL C00031 V=800.0 PL=0
MOVL C00032 V=800.0 PL=0
MOVL C00033 V=800.0 PL=0
MOVL C00034 V=800.0 PL=0
MOVL C00035 V=800.0 PL=0
MOVL C00036 V=800.0 PL=0
MOVL C00037 V=800.0 PL=0
MOVL C00038 V=800.0 PL=0
MOVL C00039 V=800.0 PL=0
MOVL C00040 V=800.0 PL=0
MOVL C00041 V=800.0 PL=0
MOVL C00042 V=800.0 PL=0
MOVL C00043 V=800.0 PL=0
MOVL C00044 V=800.0 PL=0
MOVL C00045 V=800.0 PL=0
MOVL C00046 V=800.0 PL=0
MOVL C00047 V=800.0 PL=0
MOVL C00048 V=800.0 PL=0
MOVL C00049 V=800.0 PL=0
MOVL C00050 V=800.0 PL=0
MOVL C00051 V=800.0 PL=0
MOVL C00052 V=800.0 PL=0
MOVL C00053 V=800.0 PL=0
MOVL C00054 V=800.0 PL=0
MOVL C00055 V=800.0 PL=0
MOVL C00056 V=800.0 PL=0
MOVL C00057 V=800.0 PL=0
MOVL C00058 V=800.0 PL=0
MOVL C00059 V=800.0 PL=0
MOVL C00060 V=800.0 PL=0
MOVL C00061 V=800.0 PL=0
MOVL C00062 V=800.0 PL=0
MOVL C00063 V=800.0 PL=0
MOVL C00064 V=800.0 PL=0
MOVL C00065 V=800.0 PL=0
MOVL C00066 V=800.0 PL=0
MOVL C00067 V=800.0 PL=0
MOVL C00068 V=800.0 PL=0
MOVL C00069 V=800.0 PL=0
MOVL C00070 V=800.0 PL=0
MOVL C00071 V=800.0 PL=0
MOVL C00072 V=800.0 PL=0
MOVL C00073 V=800.0 PL=0
MOVL C00074 V=800.0 PL=0
MOVL C00075 V=800.0 PL=0
MOVL C00076 V=800.0 PL=0
MOVL C00077 V=800.0 PL=0
MOVL C00078 V=800.0 PL=0
MOVL C00079 V=800.0 PL=0
MOVL C00080 V=800.0 PL=0
MOVL C00081 V=800.0 PL=0
MOVL C00082 V=800.0 PL=0
MOVL C00083 V=800.0 PL=0
MOVL C00084 V=800.0 PL=0
MOVL C00085 V=800.0 PL=0
MOVL C00086 V=800.0 PL=0
MOVL C00087 V=800.0 PL=0
MOVL C00088 V=800.0 PL=0
MOVL C00089 V=800.0 PL=0
MOVL C00090 V=800.0 PL=0
MOVL C00091 V=800.0 PL=0
MOVL C00092 V=800.0 PL=0
MOVL C00093 V=800.0 PL=0
MOVL C00094 V=800.0 PL=0
MOVL C00095 V=800.0 PL=0
MOVL C00096 V=800.0 PL=0
MOVL C00097 V=800.0 PL=0
MOVL C00098 V=800.0 PL=0
MOVL C00099 V=800.0 PL=0
MOVL C00100 V=800.0 PL=0
MOVL C00101 V=800.0 PL=0
MOVL C00102 V=800.0 PL=0
MOVL C00103 V=800.0 PL=0
MOVL C00104 V=800.0 PL=0
MOVL C00105 V=800.0 PL=0
MOVL C00106 V=800.0 PL=0
MOVL C00107 V=800.0 PL=0
MOVL C00108 V=800.0 PL=0
MOVL C00109 V=800.0 PL=0
MOVL C00110 V=800.0 PL=0
MOVL C00111 V=800.0 PL=0
MOVL C00112 V=800.0 PL=0
MOVL C00113 V=800.0 PL=0
MOVL C00114 V=800.0 PL=0
MOVL C00115 V=800.0 PL=0
MOVL C00116 V=800.0 PL=0
MOVL C00117 V=800.0 PL=0
MOVL C00118 V=800.0 PL=0
MOVL C00119 V=800.0 PL=0
MOVL C00120 V=800.0 PL=0
MOVL C00121 V=800.0 PL=0
MOVL C00122 V=800.0 PL=0
MOVL C00123 V=800.0 PL=0
MOVL C00124 V=800.0 PL=0
MOVL C00125 V=800.0 PL=0
MOVL C00126 V=800.0 PL=0
MOVL C00127 V=800.0 PL=0
MOVL C00128 V=800.0 PL=0
MOVL C00129 V=800.0 PL=0
MOVL C00130 V=800.0 PL=0
MOVL C00131 V=800.0 PL=0
MOVL C00132 V=800.0 PL=0
MOVL C00133 V=800.0 PL=0
MOVL C00134 V=800.0 PL=0
MOVL C00135 V=800.0 PL=0
MOVL C00136 V=800.0 PL=0
MOVL C00137 V=800.0 PL=0
MOVL C00138 V=800.0 PL=0
MOVL C00139 V=800.0 PL=0
MOVL C00140 V=800.0 PL=0
MOVL C00141 V=800.0 PL=0
MOVL C00142 V=800.0 PL=0
MOVL C00143 V=800.0 PL=0
MOVL C00144 V=800.0 PL=0
MOVL C00145 V=800.0 PL=0
MOVL C00146 V=800.0 PL=0
MOVL C00147 V=800.0 PL=0
MOVL C00148 V=800.0 PL=0
MOVL C00149 V=800.0 PL=0
MOVL C00150 V=800.0 PL=0
MOVL C00151 V=800.0 PL=0
MOVL C00152 V=800.0 PL=0
MOVL C00153 V=800.0 PL=0
MOVL C00154 V=800.0 PL=0
MOVL C00155 V=800.0 PL=0
MOVL C00156 V=800.0 PL=0
MOVL C00157 V=800.0 PL=0
MOVL C00158 V=800.0 PL=0
MOVL C00159 V=800.0 PL=0
MOVL C00160 V=800.0 PL=0
MOVL C00161 V=800.0 PL=0
MOVL C00162 V=800.0 PL=0
MOVL C00163 V=800.0 PL=0
MOVL C00164 V=800.0 PL=0
MOVL C00165 V=800.0 PL=0
MOVL C00166 V=800.0 PL=0
MOVL C00167 V=800.0 PL=0
MOVL C00168 V=800.0 PL=0
MOVL C00169 V=800.0 PL=0
MOVL C00170 V=800.0 PL=0
MOVL C00171 V=800.0 PL=0
MOVL C00172 V=800.0 PL=0
MOVL C00173 V=800.0 PL=0
MOVL C00174 V=800.0 PL=0
MOVL C00175 V=800.0 PL=0
MOVL C00176 V=800.0 PL=0
MOVL C00177 V=800.0 PL=0
MOVL C00178 V=800.0 PL=0
MOVL C00179 V=800.0 PL=0
MOVL C00180 V=800.0 PL=0
MOVL C00181 V=800.0 PL=0
MOVL C00182 V=800.0 PL=0
MOVL C00183 V=800.0 PL=0
MOVL C00184 V=800.0 PL=0
MOVL C00185 V=800.0 PL=0
MOVL C00186 V=800.0 PL=0
MOVL C00187 V=800.0 PL=0
MOVL C00188 V=800.0 PL=0
MOVL C00189 V=800.0 PL=0
MOVL C00190 V=800.0 PL=0
MOVL C00191 V=800.0 PL=0
MOVL C00192 V=800.0 PL=0
MOVL C00193 V=800.0 PL=0
MOVL C00194 V=800.0 PL=0
MOVL C00195 V=800.0 PL=0
MOVL C00196 V=800.0 PL=0
MOVL C00197 V=800.0 PL=0
MOVL C00198 V=800.0 PL=0
MOVL C00199 V=800.0 PL=0
MOVL C00200 V=800.0 PL=0
MOVL C00201 V=800.0 PL=0
MOVL C00202 V=800.0 PL=0
MOVL C00203 V=800.0 PL=0
MOVL C00204 V=800.0 PL=0
MOVL C00205 V=800.0 PL=0
MOVL C00206 V=800.0 PL=0
MOVL C00207 V=800.0 PL=0
MOVL C00208 V=800.0 PL=0
MOVL C00209 V=800.0 PL=0
MOVL C00210 V=800.0 PL=0
MOVL C00211 V=800.0 PL=0
MOVL C00212 V=800.0 PL=0
MOVL C00213 V=800.0 PL=0
MOVL C00214 V=800.0 PL=0
MOVL C00215 V=800.0 PL=0
MOVL C00216 V=800.0 PL=0
MOVL C00217 V=800.0 PL=0
MOVL C00218 V=800.0 PL=0
MOVL C00219 V=800.0 PL=0
MOVL C00220 V=800.0 PL=0
MOVL C00221 V=800.0 PL=0
MOVL C00222 V=800.0 PL=0
MOVL C00223 V=800.0 PL=0
MOVL C00224 V=800.0 PL=0
MOVL C00225 V=800.0 PL=0
MOVL C00226 V=800.0 PL=0
MOVL C00227 V=800.0 PL=0
MOVL C00228 V=800.0 PL=0
MOVL C00229 V=800.0 PL=0
MOVL C00230 V=800.0 PL=0
MOVL C00231 V=800.0 PL=0
MOVL C00232 V=800.0 PL=0
MOVL C00233 V=800.0 PL=0
MOVL C00234 V=800.0 PL=0
MOVL C00235 V=800.0 PL=0
MOVL C00236 V=800.0 PL=0
MOVL C00237 V=800.0 PL=0
MOVL C00238 V=800.0 PL=0
MOVL C00239 V=800.0 PL=0
MOVL C00240 V=800.0 PL=0
MOVL C00241 V=800.0 PL=0
MOVL C00242 V=800.0 PL=0
MOVL C00243 V=800.0 PL=0
MOVL C00244 V=800.0 PL=0
MOVL C00245 V=800.0 PL=0
MOVL C00246 V=800.0 PL=0
MOVL C00247 V=800.0 PL=0
MOVL C00248 V=800.0 PL=0
MOVL C00249 V=800.0 PL=0
MOVL C00250 V=800.0 PL=0
MOVL C00251 V=800.0 PL=0
MOVL C00252 V=800.0 PL=0
MOVL C00253 V=800.0 PL=0
MOVL C00254 V=800.0 PL=0
MOVL C00255 V=800.0 PL=0
MOVL C00256 V=800.0 PL=0
MOVL C00257 V=800.0 PL=0
MOVL C00258 V=800.0 PL=0
MOVL C00259 V=800.0 PL=0
MOVL C00260 V=800.0 PL=0
MOVL C00261 V=800.0 PL=0
MOVL C00262 V=800.0 PL=0
MOVL C00263 V=800.0 PL=0
MOVL C00264 V=800.0 PL=0
MOVL C00265 V=800.0 PL=0
MOVL C00266 V=800.0 PL=0
MOVL C00267 V=800.0 PL=0
MOVL C00268 V=800.0 PL=0
MOVL C00269 V=800.0 PL=0
MOVL C00270 V=800.0 PL=0
MOVL C00271 V=800.0 PL=0
MOVL C00272 V=800.0 PL=0
MOVL C00273 V=800.0 PL=0
MOVL C00274 V=800.0 PL=0
MOVL C00275 V=800.0 PL=0
MOVL C00276 V=800.0 PL=0
MOVL C00277 V=800.0 PL=0
MOVL C00278 V=800.0 PL=0
MOVL C00279 V=800.0 PL=0
MOVL C00280 V=800.0 PL=0
MOVL C00281 V=800.0 PL=0
MOVL C00282 V=800.0 PL=0
MOVL C00283 V=800.0 PL=0
MOVL C00284 V=800.0 PL=0
MOVL C00285 V=800.0 PL=0
MOVL C00286 V=800.0 PL=0
MOVL C00287 V=800.0 PL=0
MOVL C00288 V=800.0 PL=0
MOVL C00289 V=800.0 PL=0
MOVL C00290 V=800.0 PL=0
MOVL C00291 V=800.0 PL=0
MOVL C00292 V=800.0 PL=0
MOVL C00293 V=800.0 PL=0
MOVL C00294 V=800.0 PL=0
MOVL C00295 V=800.0 PL=0
MOVL C00296 V=800.0 PL=0
MOVL C00297 V=800.0 PL=0
MOVL C00298 V=800.0 PL=0
MOVL C00299 V=800.0 PL=0
MOVL C00300 V=800.0 PL=0
MOVL C00301 V=800.0 PL=0
MOVL C00302 V=800.0 PL=0
MOVL C00303 V=800.0 PL=0
MOVL C00304 V=800.0 PL=0
MOVL C00305 V=800.0 PL=0
MOVL C00306 V=800.0 PL=0
MOVL C00307 V=800.0 PL=0
MOVL C00308 V=800.0 PL=0
MOVL C00309 V=800.0 PL=0
MOVL C00310 V=800.0 PL=0
MOVL C00311 V=800.0 PL=0
MOVL C00312 V=800.0 PL=0
MOVL C00313 V=800.0 PL=0
MOVL C00314 V=800.0 PL=0
MOVL C00315 V=800.0 PL=0
MOVL C00316 V=800.0 PL=0
MOVL C00317 V=800.0 PL=0
MOVL C00318 V=800.0 PL=0
MOVL C00319 V=800.0 PL=0
MOVL C00320 V=800.0 PL=0
MOVL C00321 V=800.0 PL=0
MOVL C00322 V=800.0 PL=0
MOVL C00323 V=800.0 PL=0
MOVL C00324 V=800.0 PL=0
MOVL C00325 V=800.0 PL=0
MOVL C00326 V=800.0 PL=0
MOVL C00327 V=800.0 PL=0
MOVL C00328 V=800.0 PL=0
MOVL C00329 V=800.0 PL=0
MOVL C00330 V=800.0 PL=0
MOVL C00331 V=800.0 PL=0
MOVL C00332 V=800.0 PL=0
MOVL C00333 V=800.0 PL=0
MOVL C00334 V=800.0 PL=0
MOVL C00335 V=800.0 PL=0
MOVL C00336 V=800.0 PL=0
MOVL C00337 V=800.0 PL=0
MOVL C00338 V=800.0 PL=0
MOVL C00339 V=800.0 PL=0
MOVL C00340 V=800.0 PL=0
MOVL C00341 V=800.0 PL=0
MOVL C00342 V=800.0 PL=0
MOVL C00343 V=800.0 PL=0
MOVL C00344 V=800.0 PL=0
MOVL C00345 V=800.0 PL=0
MOVL C00346 V=800.0 PL=0
MOVL C00347 V=800.0 PL=0
MOVL C00348 V=800.0 PL=0
MOVL C00349 V=800.0 PL=0
MOVL C00350 V=800.0 PL=0
MOVL C00351 V=800.0 PL=0
MOVL C00352 V=800.0 PL=0
MOVL C00353 V=800.0 PL=0
MOVL C00354 V=800.0 PL=0
MOVL C00355 V=800.0 PL=0
MOVL C00356 V=800.0 PL=0
MOVL C00357 V=800.0 PL=0
MOVL C00358 V=800.0 PL=0
MOVL C00359 V=800.0 PL=0
MOVL C00360 V=800.0 PL=0
MOVL C00361 V=800.0 PL=0
MOVL C00362 V=800.0 PL=0
MOVL C00363 V=800.0 PL=0
MOVL C00364 V=800.0 PL=0
MOVL C00365 V=800.0 PL=0
MOVL C00366 V=800.0 PL=0
MOVL C00367 V=800.0 PL=0
MOVL C00368 V=800.0 PL=0
MOVL C00369 V=800.0 PL=0
MOVL C00370 V=800.0 PL=0
MOVL C00371 V=800.0 PL=0
MOVL C00372 V=800.0 PL=0
MOVL C00373 V=800.0 PL=0
MOVL C00374 V=800.0 PL=0
MOVL C00375 V=800.0 PL=0
MOVL C00376 V=800.0 PL=0
MOVL C00377 V=800.0 PL=0
MOVL C00378 V=800.0 PL=0
MOVL C00379 V=800.0 PL=0
MOVL C00380 V=800.0 PL=0
MOVL C00381 V=800.0 PL=0
MOVL C00382 V=800.0 PL=0
MOVL C00383 V=800.0 PL=0
MOVL C00384 V=800.0 PL=0
MOVL C00385 V=800.0 PL=0
MOVL C00386 V=800.0 PL=0
MOVL C00387 V=800.0 PL=0
MOVL C00388 V=800.0 PL=0
MOVL C00389 V=800.0 PL=0
MOVL C00390 V=800.0 PL=0
MOVL C00391 V=800.0 PL=0
MOVL C00392 V=800.0 PL=0
MOVL C00393 V=800.0 PL=0
MOVL C00394 V=800.0 PL=0
MOVL C00395 V=800.0 PL=0
MOVL C00396 V=800.0 PL=0
MOVL C00397 V=800.0 PL=0
MOVL C00398 V=800.0 PL=0
MOVL C00399 V=800.0 PL=0
MOVL C00400 V=800.0 PL=0
MOVL C00401 V=800.0 PL=0
MOVL C00402 V=800.0 PL=0
MOVL C00403 V=800.0 PL=0
MOVL C00404 V=800.0 PL=0
MOVL C00405 V=800.0 PL=0
MOVL C00406 V=800.0 PL=0
MOVL C00407 V=800.0 PL=0
MOVL C00408 V=800.0 PL=0
MOVL C00409 V=800.0 PL=0
MOVL C00410 V=800.0 PL=0
MOVL C00411 V=800.0 PL=0
MOVL C00412 V=800.0 PL=0
MOVL C00413 V=800.0 PL=0
MOVL C00414 V=800.0 PL=0
MOVL C00415 V=800.0 PL=0
MOVL C00416 V=800.0 PL=0
MOVL C00417 V=800.0 PL=0
MOVL C00418 V=800.0 PL=0
MOVL C00419 V=800.0 PL=0
MOVL C00420 V=800.0 PL=0
MOVL C00421 V=800.0 PL=0
MOVL C00422 V=800.0 PL=0
MOVL C00423 V=800.0 PL=0
MOVL C00424 V=800.0 PL=0
MOVL C00425 V=800.0 PL=0
MOVL C00426 V=800.0 PL=0
MOVL C00427 V=800.0 PL=0
MOVL C00428 V=800.0 PL=0
MOVL C00429 V=800.0 PL=0
MOVL C00430 V=800.0 PL=0
MOVL C00431 V=800.0 PL=0
MOVL C00432 V=800.0 PL=0
MOVL C00433 V=800.0 PL=0
MOVL C00434 V=800.0 PL=0
MOVL C00435 V=800.0 PL=0
MOVL C00436 V=800.0 PL=0
MOVL C00437 V=800.0 PL=0
MOVL C00438 V=800.0 PL=0
MOVL C00439 V=800.0 PL=0
MOVL C00440 V=800.0 PL=0
MOVL C00441 V=800.0 PL=0
MOVL C00442 V=800.0 PL=0
MOVL C00443 V=800.0 PL=0
MOVL C00444 V=800.0 PL=0
MOVL C00445 V=800.0 PL=0
MOVL C00446 V=800.0 PL=0
MOVL C00447 V=800.0 PL=0
MOVL C00448 V=800.0 PL=0
MOVL C00449 V=800.0 PL=0
MOVL C00450 V=800.0 PL=0
MOVL C00451 V=800.0 PL=0
MOVL C00452 V=800.0 PL=0
MOVL C00453 V=800.0 PL=0
MOVL C00454 V=800.0 PL=0
MOVL C00455 V=800.0 PL=0
MOVL C00456 V=800.0 PL=0
MOVL C00457 V=800.0 PL=0
MOVL C00458 V=800.0 PL=0
MOVL C00459 V=800.0 PL=0
MOVL C00460 V=800.0 PL=0
MOVL C00461 V=800.0 PL=0
MOVL C00462 V=800.0 PL=0
MOVL C00463 V=800.0 PL=0
MOVL C00464 V=800.0 PL=0
MOVL C00465 V=800.0 PL=0
MOVL C00466 V=800.0 PL=0
MOVL C00467 V=800.0 PL=0
MOVL C00468 V=800.0 PL=0
MOVL C00469 V=800.0 PL=0
MOVL C00470 V=800.0 PL=0
MOVL C00471 V=800.0 PL=0
MOVL C00472 V=800.0 PL=0
MOVL C00473 V=800.0 PL=0
MOVL C00474 V=800.0 PL=0
MOVL C00475 V=800.0 PL=0
MOVL C00476 V=800.0 PL=0
MOVL C00477 V=800.0 PL=0
MOVL C00478 V=800.0 PL=0
MOVL C00479 V=800.0 PL=0
MOVL C00480 V=800.0 PL=0
MOVL C00481 V=800.0 PL=0
MOVL C00482 V=800.0 PL=0
MOVL C00483 V=800.0 PL=0
MOVL C00484 V=800.0 PL=0
MOVL C00485 V=800.0 PL=0
MOVL C00486 V=800.0 PL=0
MOVL C00487 V=800.0 PL=0
MOVL C00488 V=800.0 PL=0
MOVL C00489 V=800.0 PL=0
MOVL C00490 V=800.0 PL=0
MOVL C00491 V=800.0 PL=0
MOVL C00492 V=800.0 PL=0
MOVL C00493 V=800.0 PL=0
MOVL C00494 V=800.0 PL=0
MOVL C00495 V=800.0 PL=0
MOVL C00496 V=800.0 PL=0
MOVL C00497 V=800.0 PL=0
MOVL C00498 V=800.0 PL=0
MOVL C00499 V=800.0 PL=0
MOVL C00500 V=800.0 PL=0
MOVL C00501 V=800.0 PL=0
MOVL C00502 V=800.0 PL=0
MOVL C00503 V=800.0 PL=0
MOVL C00504 V=800.0 PL=0
MOVL C00505 V=800.0 PL=0
MOVL C00506 V=800.0 PL=0
MOVL C00507 V=800.0 PL=0
MOVL C00508 V=800.0 PL=0
MOVL C00509 V=800.0 PL=0
MOVL C00510 V=800.0 PL=0
MOVL C00511 V=800.0 PL=0
MOVL C00512 V=800.0 PL=0
MOVL C00513 V=800.0 PL=0
MOVL C00514 V=800.0 PL=0
MOVL C00515 V=800.0 PL=0
MOVL C00516 V=800.0 PL=0
MOVL C00517 V=800.0 PL=0
MOVL C00518 V=800.0 PL=0
MOVL C00519 V=800.0 PL=0
MOVL C00520 V=800.0 PL=0
MOVL C00521 V=800.0 PL=0
MOVL C00522 V=800.0 PL=0
MOVL C00523 V=800.0 PL=0
MOVL C00524 V=800.0 PL=0
MOVL C00525 V=800.0 PL=0
MOVL C00526 V=800.0 PL=0
MOVL C00527 V=800.0 PL=0
MOVL C00528 V=800.0 PL=0
MOVL C00529 V=800.0 PL=0
MOVL C00530 V=800.0 PL=0
MOVL C00531 V=800.0 PL=0
MOVL C00532 V=800.0 PL=0
MOVL C00533 V=800.0 PL=0
MOVL C00534 V=800.0 PL=0
MOVL C00535 V=800.0 PL=0
MOVL C00536 V=800.0 PL=0
MOVL C00537 V=800.0 PL=0
MOVL C00538 V=800.0 PL=0
MOVL C00539 V=800.0 PL=0
MOVL C00540 V=800.0 PL=0
MOVL C00541 V=800.0 PL=0
MOVL C00542 V=800.0 PL=0
MOVL C00543 V=800.0 PL=0
MOVL C00544 V=800.0 PL=0
MOVL C00545 V=800.0 PL=0
MOVL C00546 V=800.0 PL=0
MOVL C00547 V=800.0 PL=0
MOVL C00548 V=800.0 PL=0
MOVL C00549 V=800.0 PL=0
MOVL C00550 V=800.0 PL=0
MOVL C00551 V=800.0 PL=0
MOVL C00552 V=800.0 PL=0
MOVL C00553 V=800.0 PL=0
MOVL C00554 V=800.0 PL=0
MOVL C00555 V=800.0 PL=0
MOVL C00556 V=800.0 PL=0
MOVL C00557 V=800.0 PL=0
MOVL C00558 V=800.0 PL=0
MOVL C00559 V=800.0 PL=0
MOVL C00560 V=800.0 PL=0
MOVL C00561 V=800.0 PL=0
MOVL C00562 V=800.0 PL=0
MOVL C00563 V=800.0 PL=0
MOVL C00564 V=800.0 PL=0
MOVL C00565 V=800.0 PL=0
MOVL C00566 V=800.0 PL=0
MOVL C00567 V=800.0 PL=0
MOVL C00568 V=800.0 PL=0
MOVL C00569 V=800.0 PL=0
MOVL C00570 V=800.0 PL=0
MOVL C00571 V=800.0 PL=0
MOVL C00572 V=800.0 PL=0
MOVL C00573 V=800.0 PL=0
MOVL C00574 V=800.0 PL=0
MOVL C00575 V=800.0 PL=0
MOVL C00576 V=800.0 PL=0
MOVL C00577 V=800.0 PL=0
MOVL C00578 V=800.0 PL=0
MOVL C00579 V=800.0 PL=0
MOVL C00580 V=800.0 PL=0
MOVL C00581 V=800.0 PL=0
MOVL C00582 V=800.0 PL=0
MOVL C00583 V=800.0 PL=0
MOVL C00584 V=800.0 PL=0
MOVL C00585 V=800.0 PL=0
MOVL C00586 V=800.0 PL=0
MOVL C00587 V=800.0 PL=0
MOVL C00588 V=800.0 PL=0
MOVL C00589 V=800.0 PL=0
MOVL C00590 V=800.0 PL=0
MOVL C00591 V=800.0 PL=0
MOVL C00592 V=800.0 PL=0
MOVL C00593 V=800.0 PL=0
MOVL C00594 V=800.0 PL=0
MOVL C00595 V=800.0 PL=0
MOVL C00596 V=800.0 PL=0
MOVL C00597 V=800.0 PL=0
MOVL C00598 V=800.0 PL=0
MOVL C00599 V=800.0 PL=0
MOVL C00600 V=800.0 PL=0
MOVL C00601 V=800.0 PL=0
MOVL C00602 V=800.0 PL=0
MOVL C00603 V=800.0 PL=0
MOVL C00604 V=800.0 PL=0
MOVL C00605 V=800.0 PL=0
MOVL C00606 V=800.0 PL=0
MOVL C00607 V=800.0 PL=0
MOVL C00608 V=800.0 PL=0
MOVL C00609 V=800.0 PL=0
MOVL C00610 V=800.0 PL=0
MOVL C00611 V=800.0 PL=0
MOVL C00612 V=800.0 PL=0
MOVL C00613 V=800.0 PL=0
MOVL C00614 V=800.0 PL=0
MOVL C00615 V=800.0 PL=0
MOVL C00616 V=800.0 PL=0
MOVL C00617 V=800.0 PL=0
MOVL C00618 V=800.0 PL=0
MOVL C00619 V=800.0 PL=0
MOVL C00620 V=800.0 PL=0
MOVL C00621 V=800.0 PL=0
MOVL C00622 V=800.0 PL=0
MOVL C00623 V=800.0 PL=0
MOVL C00624 V=800.0 PL=0
MOVL C00625 V=800.0 PL=0
MOVL C00626 V=800.0 PL=0
MOVL C00627 V=800.0 PL=0
MOVL C00628 V=800.0 PL=0
MOVL C00629 V=800.0 PL=0
MOVL C00630 V=800.0 PL=0
MOVL C00631 V=800.0 PL=0
MOVL C00632 V=800.0 PL=0
MOVL C00633 V=800.0 PL=0
MOVL C00634 V=800.0 PL=0
MOVL C00635 V=800.0 PL=0
MOVL C00636 V=800.0 PL=0
MOVL C00637 V=800.0 PL=0
MOVL C00638 V=800.0 PL=0
MOVL C00639 V=800.0 PL=0
MOVL C00640 V=800.0 PL=0
MOVL C00641 V=800.0 PL=0
MOVL C00642 V=800.0 PL=0
MOVL C00643 V=800.0 PL=0
MOVL C00644 V=800.0 PL=0
MOVL C00645 V=800.0 PL=0
MOVL C00646 V=800.0 PL=0
MOVL C00647 V=800.0 PL=0
MOVL C00648 V=800.0 PL=0
MOVL C00649 V=800.0 PL=0
MOVL C00650 V=800.0 PL=0
MOVL C00651 V=800.0 PL=0
MOVL C00652 V=800.0 PL=0
MOVL C00653 V=800.0 PL=0
MOVL C00654 V=800.0 PL=0
MOVL C00655 V=800.0 PL=0
MOVL C00656 V=800.0 PL=0
MOVL C00657 V=800.0 PL=0
MOVL C00658 V=800.0 PL=0
MOVL C00659 V=800.0 PL=0
MOVL C00660 V=800.0 PL=0
MOVL C00661 V=800.0 PL=0
MOVL C00662 V=800.0 PL=0
MOVL C00663 V=800.0 PL=0
MOVL C00664 V=800.0 PL=0
MOVL C00665 V=800.0 PL=0
MOVL C00666 V=800.0 PL=0
MOVL C00667 V=800.0 PL=0
MOVL C00668 V=800.0 PL=0
MOVL C00669 V=800.0 PL=0
MOVL C00670 V=800.0 PL=0
MOVL C00671 V=800.0 PL=0
MOVL C00672 V=800.0 PL=0
MOVL C00673 V=800.0 PL=0
MOVL C00674 V=800.0 PL=0
MOVL C00675 V=800.0 PL=0
MOVL C00676 V=800.0 PL=0
MOVL C00677 V=800.0 PL=0
MOVL C00678 V=800.0 PL=0
MOVL C00679 V=800.0 PL=0
MOVL C00680 V=800.0 PL=0
MOVL C00681 V=800.0 PL=0
MOVL C00682 V=800.0 PL=0
MOVL C00683 V=800.0 PL=0
MOVL C00684 V=800.0 PL=0
MOVL C00685 V=800.0 PL=0
MOVL C00686 V=800.0 PL=0
MOVL C00687 V=800.0 PL=0
MOVL C00688 V=800.0 PL=0
MOVL C00689 V=800.0 PL=0
MOVL C00690 V=800.0 PL=0
MOVL C00691 V=800.0 PL=0
MOVL C00692 V=800.0 PL=0
MOVL C00693 V=800.0 PL=0
MOVL C00694 V=800.0 PL=0
MOVL C00695 V=800.0 PL=0
MOVL C00696 V=800.0 PL=0
MOVL C00697 V=800.0 PL=0
MOVL C00698 V=800.0 PL=0
MOVL C00699 V=800.0 PL=0
MOVL C00700 V=800.0 PL=0
MOVL C00701 V=800.0 PL=0
MOVL C00702 V=800.0 PL=0
MOVL C00703 V=800.0 PL=0
MOVL C00704 V=800.0 PL=0
MOVL C00705 V=800.0 PL=0
MOVL C00706 V=800.0 PL=0
MOVL C00707 V=800.0 PL=0
MOVL C00708 V=800.0 PL=0
MOVL C00709 V=800.0 PL=0
MOVL C00710 V=800.0 PL=0
MOVL C00711 V=800.0 PL=0
MOVL C00712 V=800.0 PL=0
MOVL C00713 V=800.0 PL=0
MOVL C00714 V=800.0 PL=0
MOVL C00715 V=800.0 PL=0
MOVL C00716 V=800.0 PL=0
MOVL C00717 V=800.0 PL=0
MOVL C00718 V=800.0 PL=0
MOVL C00719 V=800.0 PL=0
MOVL C00720 V=800.0 PL=0
MOVL C00721 V=800.0 PL=0
MOVL C00722 V=800.0 PL=0
MOVL C00723 V=800.0 PL=0
MOVL C00724 V=800.0 PL=0
MOVL C00725 V=800.0 PL=0
MOVL C00726 V=800.0 PL=0
MOVL C00727 V=800.0 PL=0
MOVL C00728 V=800.0 PL=0
MOVL C00729 V=800.0 PL=0
MOVL C00730 V=800.0 PL=0
MOVL C00731 V=800.0 PL=0
MOVL C00732 V=800.0 PL=0
MOVL C00733 V=800.0 PL=0
MOVL C00734 V=800.0 PL=0
MOVL C00735 V=800.0 PL=0
MOVL C00736 V=800.0 PL=0
MOVL C00737 V=800.0 PL=0
MOVL C00738 V=800.0 PL=0
MOVL C00739 V=800.0 PL=0
MOVL C00740 V=800.0 PL=0
MOVL C00741 V=800.0 PL=0
MOVL C00742 V=800.0 PL=0
MOVL C00743 V=800.0 PL=0
MOVL C00744 V=800.0 PL=0
MOVL C00745 V=800.0 PL=0
MOVL C00746 V=800.0 PL=0
MOVL C00747 V=800.0 PL=0
MOVL C00748 V=800.0 PL=0
MOVL C00749 V=800.0 PL=0
MOVL C00750 V=800.0 PL=0
MOVL C00751 V=800.0 PL=0
MOVL C00752 V=800.0 PL=0
MOVL C00753 V=800.0 PL=0
MOVL C00754 V=800.0 PL=0
MOVL C00755 V=800.0 PL=0
MOVL C00756 V=800.0 PL=0
MOVL C00757 V=800.0 PL=0
MOVL C00758 V=800.0 PL=0
MOVL C00759 V=800.0 PL=0
MOVL C00760 V=800.0 PL=0
MOVL C00761 V=800.0 PL=0
MOVL C00762 V=800.0 PL=0
MOVL C00763 V=800.0 PL=0
MOVL C00764 V=800.0 PL=0
MOVL C00765 V=800.0 PL=0
MOVL C00766 V=800.0 PL=0
MOVL C00767 V=800.0 PL=0
MOVL C00768 V=800.0 PL=0
MOVL C00769 V=800.0 PL=0
MOVL C00770 V=800.0 PL=0
MOVL C00771 V=800.0 PL=0
MOVL C00772 V=800.0 PL=0
MOVL C00773 V=800.0 PL=0
MOVL C00774 V=800.0 PL=0
MOVL C00775 V=800.0 PL=0
MOVL C00776 V=800.0 PL=0
MOVL C00777 V=800.0 PL=0
MOVL C00778 V=800.0 PL=0
MOVL C00779 V=800.0 PL=0
MOVL C00780 V=800.0 PL=0
MOVL C00781 V=800.0 PL=0
MOVL C00782 V=800.0 PL=0
MOVL C00783 V=800.0 PL=0
MOVL C00784 V=800.0 PL=0
MOVL C00785 V=800.0 PL=0
MOVL C00786 V=800.0 PL=0
MOVL C00787 V=800.0 PL=0
MOVL C00788 V=800.0 PL=0
MOVL C00789 V=800.0 PL=0
MOVL C00790 V=800.0 PL=0
MOVL C00791 V=800.0 PL=0
MOVL C00792 V=800.0 PL=0
MOVL C00793 V=800.0 PL=0
MOVL C00794 V=800.0 PL=0
MOVL C00795 V=800.0 PL=0
MOVL C00796 V=800.0 PL=0
MOVL C00797 V=800.0 PL=0
MOVL C00798 V=800.0 PL=0
MOVL C00799 V=800.0 PL=0
MOVL C00800 V=800.0 PL=0
MOVL C00801 V=800.0 PL=0
MOVL C00802 V=800.0 PL=0
MOVL C00803 V=800.0 PL=0
MOVL C00804 V=800.0 PL=0
MOVL C00805 V=800.0 PL=0
MOVL C00806 V=800.0 PL=0
MOVL C00807 V=800.0 PL=0
MOVL C00808 V=800.0 PL=0
MOVL C00809 V=800.0 PL=0
MOVL C00810 V=800.0 PL=0
MOVL C00811 V=800.0 PL=0
MOVL C00812 V=800.0 PL=0
MOVL C00813 V=800.0 PL=0
MOVL C00814 V=800.0 PL=0
MOVL C00815 V=800.0 PL=0
MOVL C00816 V=800.0 PL=0
MOVL C00817 V=800.0 PL=0
MOVL C00818 V=800.0 PL=0
MOVL C00819 V=800.0 PL=0
MOVL C00820 V=800.0 PL=0
MOVL C00821 V=800.0 PL=0
MOVL C00822 V=800.0 PL=0
MOVL C00823 V=800.0 PL=0
MOVL C00824 V=800.0 PL=0
MOVL C00825 V=800.0 PL=0
MOVL C00826 V=800.0 PL=0
MOVL C00827 V=800.0 PL=0
MOVL C00828 V=800.0 PL=0
MOVL C00829 V=800.0 PL=0
MOVL C00830 V=800.0 PL=0
MOVL C00831 V=800.0 PL=0
MOVL C00832 V=800.0 PL=0
MOVL C00833 V=800.0 PL=0
MOVL C00834 V=800.0 PL=0
MOVL C00835 V=800.0 PL=0
MOVL C00836 V=800.0 PL=0
MOVL C00837 V=800.0 PL=0
MOVL C00838 V=800.0 PL=0
MOVL C00839 V=800.0 PL=0
MOVL C00840 V=800.0 PL=0
MOVL C00841 V=800.0 PL=0
MOVL C00842 V=800.0 PL=0
MOVL C00843 V=800.0 PL=0
MOVL C00844 V=800.0 PL=0
MOVL C00845 V=800.0 PL=0
MOVL C00846 V=800.0 PL=0
MOVL C00847 V=800.0 PL=0
MOVL C00848 V=800.0 PL=0
MOVL C00849 V=800.0 PL=0
MOVL C00850 V=800.0 PL=0
MOVL C00851 V=800.0 PL=0
MOVL C00852 V=800.0 PL=0
MOVL C00853 V=800.0 PL=0
MOVL C00854 V=800.0 PL=0
MOVL C00855 V=800.0 PL=0
MOVL C00856 V=800.0 PL=0
MOVL C00857 V=800.0 PL=0
MOVL C00858 V=800.0 PL=0
MOVL C00859 V=800.0 PL=0
MOVL C00860 V=800.0 PL=0
MOVL C00861 V=800.0 PL=0
MOVL C00862 V=800.0 PL=0
MOVL C00863 V=800.0 PL=0
MOVL C00864 V=800.0 PL=0
MOVL C00865 V=800.0 PL=0
MOVL C00866 V=800.0 PL=0
MOVL C00867 V=800.0 PL=0
MOVL C00868 V=800.0 PL=0
MOVL C00869 V=800.0 PL=0
MOVL C00870 V=800.0 PL=0
MOVL C00871 V=800.0 PL=0
MOVL C00872 V=800.0 PL=0
MOVL C00873 V=800.0 PL=0
MOVL C00874 V=800.0 PL=0
MOVL C00875 V=800.0 PL=0
MOVL C00876 V=800.0 PL=0
MOVL C00877 V=800.0 PL=0
MOVL C00878 V=800.0 PL=0
MOVL C00879 V=800.0 PL=0
MOVL C00880 V=800.0 PL=0
MOVL C00881 V=800.0 PL=0
MOVL C00882 V=800.0 PL=0
MOVL C00883 V=800.0 PL=0
MOVL C00884 V=800.0 PL=0
MOVL C00885 V=800.0 PL=0
MOVL C00886 V=800.0 PL=0
MOVL C00887 V=800.0 PL=0
MOVL C00888 V=800.0 PL=0
MOVL C00889 V=800.0 PL=0
MOVL C00890 V=800.0 PL=0
MOVL C00891 V=800.0 PL=0
MOVL C00892 V=800.0 PL=0
MOVL C00893 V=800.0 PL=0
MOVL C00894 V=800.0 PL=0
MOVL C00895 V=800.0 PL=0
MOVL C00896 V=800.0 PL=0
MOVL C00897 V=800.0 PL=0
MOVL C00898 V=800.0 PL=0
MOVL C00899 V=800.0 PL=0
MOVL C00900 V=800.0 PL=0
MOVL C00901 V=800.0 PL=0
MOVL C00902 V=800.0 PL=0
MOVL C00903 V=800.0 PL=0
MOVL C00904 V=800.0 PL=0
MOVL C00905 V=800.0 PL=0
MOVL C00906 V=800.0 PL=0
MOVL C00907 V=800.0 PL=0
MOVL C00908 V=800.0 PL=0
MOVL C00909 V=800.0 PL=0
MOVL C00910 V=800.0 PL=0
MOVL C00911 V=800.0 PL=0
MOVL C00912 V=800.0 PL=0
MOVL C00913 V=800.0 PL=0
MOVL C00914 V=800.0 PL=0
MOVL C00915 V=800.0 PL=0
MOVL C00916 V=800.0 PL=0
MOVL C00917 V=800.0 PL=0
MOVL C00918 V=800.0 PL=0
MOVL C00919 V=800.0 PL=0
MOVL C00920 V=800.0 PL=0
MOVL C00921 V=800.0 PL=0
MOVL C00922 V=800.0 PL=0
MOVL C00923 V=800.0 PL=0
MOVL C00924 V=800.0 PL=0
MOVL C00925 V=800.0 PL=0
MOVL C00926 V=800.0 PL=0
MOVL C00927 V=800.0 PL=0
MOVL C00928 V=800.0 PL=0
MOVL C00929 V=800.0 PL=0
MOVL C00930 V=800.0 PL=0
MOVL C00931 V=800.0 PL=0
MOVL C00932 V=800.0 PL=0
MOVL C00933 V=800.0 PL=0
MOVL C00934 V=800.0 PL=0
MOVL C00935 V=800.0 PL=0
MOVL C00936 V=800.0 PL=0
MOVL C00937 V=800.0 PL=0
MOVL C00938 V=800.0 PL=0
MOVL C00939 V=800.0 PL=0
MOVL C00940 V=800.0 PL=0
MOVL C00941 V=800.0 PL=0
MOVL C00942 V=800.0 PL=0
MOVL C00943 V=800.0 PL=0
MOVL C00944 V=800.0 PL=0
MOVL C00945 V=800.0 PL=0
MOVL C00946 V=800.0 PL=0
MOVL C00947 V=800.0 PL=0
MOVL C00948 V=800.0 PL=0
MOVL C00949 V=800.0 PL=0
MOVL C00950 V=800.0 PL=0
MOVL C00951 V=800.0 PL=0
MOVL C00952 V=800.0 PL=0
MOVL C00953 V=800.0 PL=0
MOVL C00954 V=800.0 PL=0
MOVL C00955 V=800.0 PL=0
MOVL C00956 V=800.0 PL=0
MOVL C00957 V=800.0 PL=0
MOVL C00958 V=800.0 PL=0
MOVL C00959 V=800.0 PL=0
MOVL C00960 V=800.0 PL=0
MOVL C00961 V=800.0 PL=0
MOVL C00962 V=800.0 PL=0
MOVL C00963 V=800.0 PL=0
MOVL C00964 V=800.0 PL=0
MOVL C00965 V=800.0 PL=0
MOVL C00966 V=800.0 PL=0
MOVL C00967 V=800.0 PL=0
MOVL C00968 V=800.0 PL=0
MOVL C00969 V=800.0 PL=0
MOVL C00970 V=800.0 PL=0
MOVL C00971 V=800.0 PL=0
MOVL C00972 V=800.0 PL=0
MOVL C00973 V=800.0 PL=0
MOVL C00974 V=800.0 PL=0
MOVL C00975 V=800.0 PL=0
MOVL C00976 V=800.0 PL=0
MOVL C00977 V=800.0 PL=0
MOVL C00978 V=800.0 PL=0
MOVL C00979 V=800.0 PL=0
MOVL C00980 V=800.0 PL=0
MOVL C00981 V=800.0 PL=0
MOVL C00982 V=800.0 PL=0
MOVL C00983 V=800.0 PL=0
MOVL C00984 V=800.0 PL=0
MOVL C00985 V=800.0 PL=0
MOVL C00986 V=800.0 PL=0
MOVL C00987 V=800.0 PL=0
MOVL C00988 V=800.0 PL=0
MOVL C00989 V=800.0 PL=0
MOVL C00990 V=800.0 PL=0
MOVL C00991 V=800.0 PL=0
MOVL C00992 V=800.0 PL=0
MOVL C00993 V=800.0 PL=0
MOVL C00994 V=800.0 PL=0
MOVL C00995 V=800.0 PL=0
MOVL C00996 V=800.0 PL=0
MOVL C00997 V=800.0 PL=0
MOVL C00998 V=800.0 PL=0
MOVL C00999 V=800.0 PL=0
MOVL C01000 V=800.0 PL=0
MOVL C01001 V=800.0 PL=0
MOVL C01002 V=800.0 PL=0
MOVL C01003 V=800.0 PL=0
MOVL C01004 V=800.0 PL=0
MOVL C01005 V=800.0 PL=0
MOVL C01006 V=800.0 PL=0
MOVL C01007 V=800.0 PL=0
MOVL C01008 V=800.0 PL=0
MOVL C01009 V=800.0 PL=0
MOVL C01010 V=800.0 PL=0
MOVL C01011 V=800.0 PL=0
MOVL C01012 V=800.0 PL=0
MOVL C01013 V=800.0 PL=0
MOVL C01014 V=800.0 PL=0
MOVL C01015 V=800.0 PL=0
MOVL C01016 V=800.0 PL=0
MOVL C01017 V=800.0 PL=0
MOVL C01018 V=800.0 PL=0
MOVL C01019 V=800.0 PL=0
MOVL C01020 V=800.0 PL=0
MOVL C01021 V=800.0 PL=0
MOVL C01022 V=800.0 PL=0
MOVL C01023 V=800.0 PL=0
MOVL C01024 V=800.0 PL=0
MOVL C01025 V=800.0 PL=0
MOVL C01026 V=800.0 PL=0
MOVL C01027 V=800.0 PL=0
MOVL C01028 V=800.0 PL=0
MOVL C01029 V=800.0 PL=0
MOVL C01030 V=800.0 PL=0
MOVL C01031 V=800.0 PL=0
MOVL C01032 V=800.0 PL=0
MOVL C01033 V=800.0 PL=0
MOVL C01034 V=800.0 PL=0
MOVL C01035 V=800.0 PL=0
MOVL C01036 V=800.0 PL=0
MOVL C01037 V=800.0 PL=0
MOVL C01038 V=800.0 PL=0
MOVL C01039 V=800.0 PL=0
MOVL C01040 V=800.0 PL=0
MOVL C01041 V=800.0 PL=0
MOVL C01042 V=800.0 PL=0
MOVL C01043 V=800.0 PL=0
MOVL C01044 V=800.0 PL=0
MOVL C01045 V=800.0 PL=0
MOVL C01046 V=800.0 PL=0
MOVL C01047 V=800.0 PL=0
MOVL C01048 V=800.0 PL=0
MOVL C01049 V=800.0 PL=0
MOVL C01050 V=800.0 PL=0
MOVL C01051 V=800.0 PL=0
MOVL C01052 V=800.0 PL=0
MOVL C01053 V=800.0 PL=0
MOVL C01054 V=800.0 PL=0
MOVL C01055 V=800.0 PL=0
MOVL C01056 V=800.0 PL=0
MOVL C01057 V=800.0 PL=0
MOVL C01058 V=800.0 PL=0
MOVL C01059 V=800.0 PL=0
MOVL C01060 V=800.0 PL=0
MOVL C01061 V=800.0 PL=0
MOVL C01062 V=800.0 PL=0
MOVL C01063 V=800.0 PL=0
MOVL C01064 V=800.0 PL=0
MOVL C01065 V=800.0 PL=0
MOVL C01066 V=800.0 PL=0
MOVL C01067 V=800.0 PL=0
MOVL C01068 V=800.0 PL=0
MOVL C01069 V=800.0 PL=0
MOVL C01070 V=800.0 PL=0
MOVL C01071 V=800.0 PL=0
MOVL C01072 V=800.0 PL=0
MOVL C01073 V=800.0 PL=0
MOVL C01074 V=800.0 PL=0
MOVL C01075 V=800.0 PL=0
MOVL C01076 V=800.0 PL=0
MOVL C01077 V=800.0 PL=0
MOVL C01078 V=800.0 PL=0
MOVL C01079 V=800.0 PL=0
MOVL C01080 V=800.0 PL=0
MOVL C01081 V=800.0 PL=0
MOVL C01082 V=800.0 PL=0
MOVL C01083 V=800.0 PL=0
MOVL C01084 V=800.0 PL=0
MOVL C01085 V=800.0 PL=0
MOVL C01086 V=800.0 PL=0
MOVL C01087 V=800.0 PL=0
MOVL C01088 V=800.0 PL=0
MOVL C01089 V=800.0 PL=0
MOVL C01090 V=800.0 PL=0
MOVL C01091 V=800.0 PL=0
MOVL C01092 V=800.0 PL=0
MOVL C01093 V=800.0 PL=0
MOVL C01094 V=800.0 PL=0
MOVL C01095 V=800.0 PL=0
MOVL C01096 V=800.0 PL=0
MOVL C01097 V=800.0 PL=0
MOVL C01098 V=800.0 PL=0
MOVL C01099 V=800.0 PL=0
MOVL C01100 V=800.0 PL=0
MOVL C01101 V=800.0 PL=0
MOVL C01102 V=800.0 PL=0
MOVL C01103 V=800.0 PL=0
MOVL C01104 V=800.0 PL=0
MOVL C01105 V=800.0 PL=0
MOVL C01106 V=800.0 PL=0
MOVL C01107 V=800.0 PL=0
MOVL C01108 V=800.0 PL=0
MOVL C01109 V=800.0 PL=0
MOVL C01110 V=800.0 PL=0
MOVL C01111 V=800.0 PL=0
MOVL C01112 V=800.0 PL=0
MOVL C01113 V=800.0 PL=0
MOVL C01114 V=800.0 PL=0
MOVL C01115 V=800.0 PL=0
MOVL C01116 V=800.0 PL=0
MOVL C01117 V=800.0 PL=0
MOVL C01118 V=800.0 PL=0
MOVL C01119 V=800.0 PL=0
MOVL C01120 V=800.0 PL=0
MOVL C01121 V=800.0 PL=0
MOVL C01122 V=800.0 PL=0
MOVL C01123 V=800.0 PL=0
MOVL C01124 V=800.0 PL=0
MOVL C01125 V=800.0 PL=0
MOVL C01126 V=800.0 PL=0
MOVL C01127 V=800.0 PL=0
MOVL C01128 V=800.0 PL=0
MOVL C01129 V=800.0 PL=0
MOVL C01130 V=800.0 PL=0
MOVL C01131 V=800.0 PL=0
MOVL C01132 V=800.0 PL=0
MOVL C01133 V=800.0 PL=0
MOVL C01134 V=800.0 PL=0
MOVL C01135 V=800.0 PL=0
MOVL C01136 V=800.0 PL=0
MOVL C01137 V=800.0 PL=0
MOVL C01138 V=800.0 PL=0
MOVL C01139 V=800.0 PL=0
MOVL C01140 V=800.0 PL=0
MOVL C01141 V=800.0 PL=0
MOVL C01142 V=800.0 PL=0
MOVL C01143 V=800.0 PL=0
MOVL C01144 V=800.0 PL=0
MOVL C01145 V=800.0 PL=0
MOVL C01146 V=800.0 PL=0
MOVL C01147 V=800.0 PL=0
MOVL C01148 V=800.0 PL=0
MOVL C01149 V=800.0 PL=0
MOVL C01150 V=800.0 PL=0
MOVL C01151 V=800.0 PL=0
MOVL C01152 V=800.0 PL=0
MOVL C01153 V=800.0 PL=0
MOVL C01154 V=800.0 PL=0
MOVL C01155 V=800.0 PL=0
MOVL C01156 V=800.0 PL=0
MOVL C01157 V=800.0 PL=0
MOVL C01158 V=800.0 PL=0
MOVL C01159 V=800.0 PL=0
MOVL C01160 V=800.0 PL=0
MOVL C01161 V=800.0 PL=0
MOVL C01162 V=800.0 PL=0
MOVL C01163 V=800.0 PL=0
MOVL C01164 V=800.0 PL=0
MOVL C01165 V=800.0 PL=0
MOVL C01166 V=800.0 PL=0
MOVL C01167 V=800.0 PL=0
MOVL C01168 V=800.0 PL=0
MOVL C01169 V=800.0 PL=0
MOVL C01170 V=800.0 PL=0
MOVL C01171 V=800.0 PL=0
MOVL C01172 V=800.0 PL=0
MOVL C01173 V=800.0 PL=0
MOVL C01174 V=800.0 PL=0
MOVL C01175 V=800.0 PL=0
MOVL C01176 V=800.0 PL=0
MOVL C01177 V=800.0 PL=0
MOVL C01178 V=800.0 PL=0
MOVL C01179 V=800.0 PL=0
MOVL C01180 V=800.0 PL=0
MOVL C01181 V=800.0 PL=0
MOVL C01182 V=800.0 PL=0
MOVL C01183 V=800.0 PL=0
MOVL C01184 V=800.0 PL=0
MOVL C01185 V=800.0 PL=0
MOVL C01186 V=800.0 PL=0
MOVL C01187 V=800.0 PL=0
MOVL C01188 V=800.0 PL=0
MOVL C01189 V=800.0 PL=0
MOVL C01190 V=800.0 PL=0
MOVL C01191 V=800.0 PL=0
MOVL C01192 V=800.0 PL=0
MOVL C01193 V=800.0 PL=0
MOVL C01194 V=800.0 PL=0
MOVL C01195 V=800.0 PL=0
MOVL C01196 V=800.0 PL=0
MOVL C01197 V=800.0 PL=0
MOVL C01198 V=800.0 PL=0
MOVL C01199 V=800.0 PL=0
MOVL C01200 V=800.0 PL=0
MOVL C01201 V=800.0 PL=0
MOVL C01202 V=800.0 PL=0
MOVL C01203 V=800.0 PL=0
MOVL C01204 V=800.0 PL=0
MOVL C01205 V=800.0 PL=0
MOVL C01206 V=800.0 PL=0
MOVL C01207 V=800.0 PL=0
MOVL C01208 V=800.0 PL=0
MOVL C01209 V=800.0 PL=0
MOVL C01210 V=800.0 PL=0
MOVL C01211 V=800.0 PL=0
MOVL C01212 V=800.0 PL=0
MOVL C01213 V=800.0 PL=0
MOVL C01214 V=800.0 PL=0
MOVL C01215 V=800.0 PL=0
MOVL C01216 V=800.0 PL=0
MOVL C01217 V=800.0 PL=0
MOVL C01218 V=800.0 PL=0
MOVL C01219 V=800.0 PL=0
MOVL C01220 V=800.0 PL=0
MOVL C01221 V=800.0 PL=0
MOVL C01222 V=800.0 PL=0
MOVL C01223 V=800.0 PL=0
MOVL C01224 V=800.0 PL=0
MOVL C01225 V=800.0 PL=0
MOVL C01226 V=800.0 PL=0
MOVL C01227 V=800.0 PL=0
MOVL C01228 V=800.0 PL=0
MOVL C01229 V=800.0 PL=0
MOVL C01230 V=800.0 PL=0
MOVL C01231 V=800.0 PL=0
MOVL C01232 V=800.0 PL=0
MOVL C01233 V=800.0 PL=0
MOVL C01234 V=800.0 PL=0
MOVL C01235 V=800.0 PL=0
MOVL C01236 V=800.0 PL=0
MOVL C01237 V=800.0 PL=0
MOVL C01238 V=800.0 PL=0
MOVL C01239 V=800.0 PL=0
MOVL C01240 V=800.0 PL=0
MOVL C01241 V=800.0 PL=0
MOVL C01242 V=800.0 PL=0
MOVL C01243 V=800.0 PL=0
MOVL C01244 V=800.0 PL=0
MOVL C01245 V=800.0 PL=0
MOVL C01246 V=800.0 PL=0
MOVL C01247 V=800.0 PL=0
MOVL C01248 V=800.0 PL=0
MOVL C01249 V=800.0 PL=0
MOVL C01250 V=800.0 PL=0
MOVL C01251 V=800.0 PL=0
MOVL C01252 V=800.0 PL=0
MOVL C01253 V=800.0 PL=0
MOVL C01254 V=800.0 PL=0
MOVL C01255 V=800.0 PL=0
MOVL C01256 V=800.0 PL=0
MOVL C01257 V=800.0 PL=0
MOVL C01258 V=800.0 PL=0
MOVL C01259 V=800.0 PL=0
MOVL C01260 V=800.0 PL=0
MOVL C01261 V=800.0 PL=0
MOVL C01262 V=800.0 PL=0
MOVL C01263 V=800.0 PL=0
MOVL C01264 V=800.0 PL=0
MOVL C01265 V=800.0 PL=0
MOVL C01266 V=800.0 PL=0
MOVL C01267 V=800.0 PL=0
MOVL C01268 V=800.0 PL=0
MOVL C01269 V=800.0 PL=0
MOVL C01270 V=800.0 PL=0
MOVL C01271 V=800.0 PL=0
MOVL C01272 V=800.0 PL=0
MOVL C01273 V=800.0 PL=0
MOVL C01274 V=800.0 PL=0
MOVL C01275 V=800.0 PL=0
MOVL C01276 V=800.0 PL=0
MOVL C01277 V=800.0 PL=0
MOVL C01278 V=800.0 PL=0
MOVL C01279 V=800.0 PL=0
MOVL C01280 V=800.0 PL=0
MOVL C01281 V=800.0 PL=0
MOVL C01282 V=800.0 PL=0
MOVL C01283 V=800.0 PL=0
MOVL C01284 V=800.0 PL=0
MOVL C01285 V=800.0 PL=0
MOVL C01286 V=800.0 PL=0
MOVL C01287 V=800.0 PL=0
MOVL C01288 V=800.0 PL=0
MOVL C01289 V=800.0 PL=0
MOVL C01290 V=800.0 PL=0
MOVL C01291 V=800.0 PL=0
MOVL C01292 V=800.0 PL=0
MOVL C01293 V=800.0 PL=0
MOVL C01294 V=800.0 PL=0
MOVL C01295 V=800.0 PL=0
MOVL C01296 V=800.0 PL=0
MOVL C01297 V=800.0 PL=0
MOVL C01298 V=800.0 PL=0
MOVL C01299 V=800.0 PL=0
MOVL C01300 V=800.0 PL=0
MOVL C01301 V=800.0 PL=0
MOVL C01302 V=800.0 PL=0
MOVL C01303 V=800.0 PL=0
MOVL C01304 V=800.0 PL=0
MOVL C01305 V=800.0 PL=0
MOVL C01306 V=800.0 PL=0
MOVL C01307 V=800.0 PL=0
MOVL C01308 V=800.0 PL=0
MOVL C01309 V=800.0 PL=0
MOVL C01310 V=800.0 PL=0
MOVL C01311 V=800.0 PL=0
MOVL C01312 V=800.0 PL=0
MOVL C01313 V=800.0 PL=0
MOVL C01314 V=800.0 PL=0
MOVL C01315 V=800.0 PL=0
MOVL C01316 V=800.0 PL=0
MOVL C01317 V=800.0 PL=0
MOVL C01318 V=800.0 PL=0
MOVL C01319 V=800.0 PL=0
MOVL C01320 V=800.0 PL=0
MOVL C01321 V=800.0 PL=0
MOVL C01322 V=800.0 PL=0
MOVL C01323 V=800.0 PL=0
MOVL C01324 V=800.0 PL=0
MOVL C01325 V=800.0 PL=0
MOVL C01326 V=800.0 PL=0
MOVL C01327 V=800.0 PL=0
MOVL C01328 V=800.0 PL=0
MOVL C01329 V=800.0 PL=0
MOVL C01330 V=800.0 PL=0
MOVL C01331 V=800.0 PL=0
MOVL C01332 V=800.0 PL=0
MOVL C01333 V=800.0 PL=0
MOVL C01334 V=800.0 PL=0
MOVL C01335 V=800.0 PL=0
MOVL C01336 V=800.0 PL=0
MOVL C01337 V=800.0 PL=0
MOVL C01338 V=800.0 PL=0
MOVL C01339 V=800.0 PL=0
MOVL C01340 V=800.0 PL=0
MOVL C01341 V=800.0 PL=0
MOVL C01342 V=800.0 PL=0
MOVL C01343 V=800.0 PL=0
MOVL C01344 V=800.0 PL=0
MOVL C01345 V=800.0 PL=0
MOVL C01346 V=800.0 PL=0
MOVL C01347 V=800.0 PL=0
MOVL C01348 V=800.0 PL=0
MOVL C01349 V=800.0 PL=0
MOVL C01350 V=800.0 PL=0
MOVL C01351 V=800.0 PL=0
MOVL C01352 V=800.0 PL=0
MOVL C01353 V=800.0 PL=0
MOVL C01354 V=800.0 PL=0
MOVL C01355 V=800.0 PL=0
MOVL C01356 V=800.0 PL=0
MOVL C01357 V=800.0 PL=0
MOVL C01358 V=800.0 PL=0
MOVL C01359 V=800.0 PL=0
MOVL C01360 V=800.0 PL=0
MOVL C01361 V=800.0 PL=0
MOVL C01362 V=800.0 PL=0
MOVL C01363 V=800.0 PL=0
MOVL C01364 V=800.0 PL=0
MOVL C01365 V=800.0 PL=0
MOVL C01366 V=800.0 PL=0
MOVL C01367 V=800.0 PL=0
MOVL C01368 V=800.0 PL=0
MOVL C01369 V=800.0 PL=0
MOVL C01370 V=800.0 PL=0
MOVL C01371 V=800.0 PL=0
MOVL C01372 V=800.0 PL=0
MOVL C01373 V=800.0 PL=0
MOVL C01374 V=800.0 PL=0
MOVL C01375 V=800.0 PL=0
MOVL C01376 V=800.0 PL=0
MOVL C01377 V=800.0 PL=0
MOVL C01378 V=800.0 PL=0
MOVL C01379 V=800.0 PL=0
MOVL C01380 V=800.0 PL=0
MOVL C01381 V=800.0 PL=0
MOVL C01382 V=800.0 PL=0
MOVL C01383 V=800.0 PL=0
MOVL C01384 V=800.0 PL=0
MOVL C01385 V=800.0 PL=0
MOVL C01386 V=800.0 PL=0
MOVL C01387 V=800.0 PL=0
MOVL C01388 V=800.0 PL=0
MOVL C01389 V=800.0 PL=0
MOVL C01390 V=800.0 PL=0
MOVL C01391 V=800.0 PL=0
MOVL C01392 V=800.0 PL=0
MOVL C01393 V=800.0 PL=0
MOVL C01394 V=800.0 PL=0
MOVL C01395 V=800.0 PL=0
MOVL C01396 V=800.0 PL=0
MOVL C01397 V=800.0 PL=0
MOVL C01398 V=800.0 PL=0
MOVL C01399 V=800.0 PL=0
MOVL C01400 V=800.0 PL=0
MOVL C01401 V=800.0 PL=0
MOVL C01402 V=800.0 PL=0
MOVL C01403 V=800.0 PL=0
MOVL C01404 V=800.0 PL=0
MOVL C01405 V=800.0 PL=0
MOVL C01406 V=800.0 PL=0
MOVL C01407 V=800.0 PL=0
MOVL C01408 V=800.0 PL=0
MOVL C01409 V=800.0 PL=0
MOVL C01410 V=800.0 PL=0
MOVL C01411 V=800.0 PL=0
MOVL C01412 V=800.0 PL=0
MOVL C01413 V=800.0 PL=0
MOVL C01414 V=800.0 PL=0
MOVL C01415 V=800.0 PL=0
MOVL C01416 V=800.0 PL=0
MOVL C01417 V=800.0 PL=0
MOVL C01418 V=800.0 PL=0
MOVL C01419 V=800.0 PL=0
MOVL C01420 V=800.0 PL=0
MOVL C01421 V=800.0 PL=0
MOVL C01422 V=800.0 PL=0
MOVL C01423 V=800.0 PL=0
MOVL C01424 V=800.0 PL=0
MOVL C01425 V=800.0 PL=0
MOVL C01426 V=800.0 PL=0
MOVL C01427 V=800.0 PL=0
MOVL C01428 V=800.0 PL=0
MOVL C01429 V=800.0 PL=0
MOVL C01430 V=800.0 PL=0
MOVL C01431 V=800.0 PL=0
MOVL C01432 V=800.0 PL=0
MOVL C01433 V=800.0 PL=0
MOVL C01434 V=800.0 PL=0
MOVL C01435 V=800.0 PL=0
MOVL C01436 V=800.0 PL=0
MOVL C01437 V=800.0 PL=0
MOVL C01438 V=800.0 PL=0
MOVL C01439 V=800.0 PL=0
MOVL C01440 V=800.0 PL=0
MOVL C01441 V=800.0 PL=0
MOVL C01442 V=800.0 PL=0
MOVL C01443 V=800.0 PL=0
MOVL C01444 V=800.0 PL=0
MOVL C01445 V=800.0 PL=0
MOVL C01446 V=800.0 PL=0
MOVL C01447 V=800.0 PL=0
MOVL C01448 V=800.0 PL=0
MOVL C01449 V=800.0 PL=0
MOVL C01450 V=800.0 PL=0
MOVL C01451 V=800.0 PL=0
MOVL C01452 V=800.0 PL=0
MOVL C01453 V=800.0 PL=0
MOVL C01454 V=800.0 PL=0
MOVL C01455 V=800.0 PL=0
MOVL C01456 V=800.0 PL=0
MOVL C01457 V=800.0 PL=0
MOVL C01458 V=800.0 PL=0
MOVL C01459 V=800.0 PL=0
MOVL C01460 V=800.0 PL=0
MOVL C01461 V=800.0 PL=0
MOVL C01462 V=800.0 PL=0
MOVL C01463 V=800.0 PL=0
MOVL C01464 V=800.0 PL=0
MOVL C01465 V=800.0 PL=0
MOVL C01466 V=800.0 PL=0
MOVL C01467 V=800.0 PL=0
MOVL C01468 V=800.0 PL=0
MOVL C01469 V=800.0 PL=0
MOVL C01470 V=800.0 PL=0
MOVL C01471 V=800.0 PL=0
MOVL C01472 V=800.0 PL=0
MOVL C01473 V=800.0 PL=0
MOVL C01474 V=800.0 PL=0
MOVL C01475 V=800.0 PL=0
MOVL C01476 V=800.0 PL=0
MOVL C01477 V=800.0 PL=0
MOVL C01478 V=800.0 PL=0
MOVL C01479 V=800.0 PL=0
MOVL C01480 V=800.0 PL=0
MOVL C01481 V=800.0 PL=0
MOVL C01482 V=800.0 PL=0
MOVL C01483 V=800.0 PL=0
MOVL C01484 V=800.0 PL=0
MOVL C01485 V=800.0 PL=0
MOVL C01486 V=800.0 PL=0
MOVL C01487 V=800.0 PL=0
MOVL C01488 V=800.0 PL=0
MOVL C01489 V=800.0 PL=0
MOVL C01490 V=800.0 PL=0
MOVL C01491 V=800.0 PL=0
MOVL C01492 V=800.0 PL=0
MOVL C01493 V=800.0 PL=0
MOVL C01494 V=800.0 PL=0
MOVL C01495 V=800.0 PL=0
MOVL C01496 V=800.0 PL=0
MOVL C01497 V=800.0 PL=0
MOVL C01498 V=800.0 PL=0
MOVL C01499 V=800.0 PL=0
MOVL C01500 V=800.0 PL=0
MOVL C01501 V=800.0 PL=0
MOVL C01502 V=800.0 PL=0
MOVL C01503 V=800.0 PL=0
MOVL C01504 V=800.0 PL=0
MOVL C01505 V=800.0 PL=0
MOVL C01506 V=800.0 PL=0
MOVL C01507 V=800.0 PL=0
MOVL C01508 V=800.0 PL=0
MOVL C01509 V=800.0 PL=0
MOVL C01510 V=800.0 PL=0
MOVL C01511 V=800.0 PL=0
MOVL C01512 V=800.0 PL=0
MOVL C01513 V=800.0 PL=0
MOVL C01514 V=800.0 PL=0
MOVL C01515 V=800.0 PL=0
MOVL C01516 V=800.0 PL=0
MOVL C01517 V=800.0 PL=0
MOVL C01518 V=800.0 PL=0
MOVL C01519 V=800.0 PL=0
MOVL C01520 V=800.0 PL=0
MOVL C01521 V=800.0 PL=0
MOVL C01522 V=800.0 PL=0
MOVL C01523 V=800.0 PL=0
MOVL C01524 V=800.0 PL=0
MOVL C01525 V=800.0 PL=0
MOVL C01526 V=800.0 PL=0
MOVL C01527 V=800.0 PL=0
MOVL C01528 V=800.0 PL=0
MOVL C01529 V=800.0 PL=0
MOVL C01530 V=800.0 PL=0
MOVL C01531 V=800.0 PL=0
MOVL C01532 V=800.0 PL=0
MOVL C01533 V=800.0 PL=0
MOVL C01534 V=800.0 PL=0
MOVL C01535 V=800.0 PL=0
MOVL C01536 V=800.0 PL=0
MOVL C01537 V=800.0 PL=0
MOVL C01538 V=800.0 PL=0
MOVL C01539 V=800.0 PL=0
MOVL C01540 V=800.0 PL=0
MOVL C01541 V=800.0 PL=0
MOVL C01542 V=800.0 PL=0
MOVL C01543 V=800.0 PL=0
MOVL C01544 V=800.0 PL=0
MOVL C01545 V=800.0 PL=0
MOVL C01546 V=800.0 PL=0
MOVL C01547 V=800.0 PL=0
MOVL C01548 V=800.0 PL=0
MOVL C01549 V=800.0 PL=0
MOVL C01550 V=800.0 PL=0
MOVL C01551 V=800.0 PL=0
MOVL C01552 V=800.0 PL=0
MOVL C01553 V=800.0 PL=0
MOVL C01554 V=800.0 PL=0
MOVL C01555 V=800.0 PL=0
MOVL C01556 V=800.0 PL=0
MOVL C01557 V=800.0 PL=0
MOVL C01558 V=800.0 PL=0
MOVL C01559 V=800.0 PL=0
MOVL C01560 V=800.0 PL=0
MOVL C01561 V=800.0 PL=0
MOVL C01562 V=800.0 PL=0
MOVL C01563 V=800.0 PL=0
MOVL C01564 V=800.0 PL=0
MOVL C01565 V=800.0 PL=0
MOVL C01566 V=800.0 PL=0
MOVL C01567 V=800.0 PL=0
MOVL C01568 V=800.0 PL=0
MOVL C01569 V=800.0 PL=0
MOVL C01570 V=800.0 PL=0
MOVL C01571 V=800.0 PL=0
MOVL C01572 V=800.0 PL=0
MOVL C01573 V=800.0 PL=0
MOVL C01574 V=800.0 PL=0
MOVL C01575 V=800.0 PL=0
MOVL C01576 V=800.0 PL=0
MOVL C01577 V=800.0 PL=0
MOVL C01578 V=800.0 PL=0
MOVL C01579 V=800.0 PL=0
MOVL C01580 V=800.0 PL=0
MOVL C01581 V=800.0 PL=0
MOVL C01582 V=800.0 PL=0
MOVL C01583 V=800.0 PL=0
MOVL C01584 V=800.0 PL=0
MOVL C01585 V=800.0 PL=0
MOVL C01586 V=800.0 PL=0
MOVL C01587 V=800.0 PL=0
MOVL C01588 V=800.0 PL=0
MOVL C01589 V=800.0 PL=0
MOVL C01590 V=800.0 PL=0
MOVL C01591 V=800.0 PL=0
MOVL C01592 V=800.0 PL=0
MOVL C01593 V=800.0 PL=0
MOVL C01594 V=800.0 PL=0
MOVL C01595 V=800.0 PL=0
MOVL C01596 V=800.0 PL=0
MOVL C01597 V=800.0 PL=0
MOVL C01598 V=800.0 PL=0
MOVL C01599 V=800.0 PL=0
MOVL C01600 V=800.0 PL=0
MOVL C01601 V=800.0 PL=0
MOVL C01602 V=800.0 PL=0
MOVL C01603 V=800.0 PL=0
MOVL C01604 V=800.0 PL=0
MOVL C01605 V=800.0 PL=0
MOVL C01606 V=800.0 PL=0
MOVL C01607 V=800.0 PL=0
MOVL C01608 V=800.0 PL=0
MOVL C01609 V=800.0 PL=0
MOVL C01610 V=800.0 PL=0
MOVL C01611 V=800.0 PL=0
MOVL C01612 V=800.0 PL=0
MOVL C01613 V=800.0 PL=0
MOVL C01614 V=800.0 PL=0
MOVL C01615 V=800.0 PL=0
MOVL C01616 V=800.0 PL=0
MOVL C01617 V=800.0 PL=0
MOVL C01618 V=800.0 PL=0
MOVL C01619 V=800.0 PL=0
MOVL C01620 V=800.0 PL=0
MOVL C01621 V=800.0 PL=0
MOVL C01622 V=800.0 PL=0
MOVL C01623 V=800.0 PL=0
MOVL C01624 V=800.0 PL=0
MOVL C01625 V=800.0 PL=0
MOVL C01626 V=800.0 PL=0
MOVL C01627 V=800.0 PL=0
MOVL C01628 V=800.0 PL=0
MOVL C01629 V=800.0 PL=0
MOVL C01630 V=800.0 PL=0
MOVL C01631 V=800.0 PL=0
MOVL C01632 V=800.0 PL=0
MOVL C01633 V=800.0 PL=0
MOVL C01634 V=800.0 PL=0
MOVL C01635 V=800.0 PL=0
MOVL C01636 V=800.0 PL=0
MOVL C01637 V=800.0 PL=0
MOVL C01638 V=800.0 PL=0
MOVL C01639 V=800.0 PL=0
MOVL C01640 V=800.0 PL=0
MOVL C01641 V=800.0 PL=0
MOVL C01642 V=800.0 PL=0
MOVL C01643 V=800.0 PL=0
MOVL C01644 V=800.0 PL=0
MOVL C01645 V=800.0 PL=0
MOVL C01646 V=800.0 PL=0
MOVL C01647 V=800.0 PL=0
MOVL C01648 V=800.0 PL=0
MOVL C01649 V=800.0 PL=0
MOVL C01650 V=800.0 PL=0
MOVL C01651 V=800.0 PL=0
MOVL C01652 V=800.0 PL=0
MOVL C01653 V=800.0 PL=0
MOVL C01654 V=800.0 PL=0
MOVL C01655 V=800.0 PL=0
MOVL C01656 V=800.0 PL=0
MOVL C01657 V=800.0 PL=0
MOVL C01658 V=800.0 PL=0
MOVL C01659 V=800.0 PL=0
MOVL C01660 V=800.0 PL=0
MOVL C01661 V=800.0 PL=0
MOVL C01662 V=800.0 PL=0
MOVL C01663 V=800.0 PL=0
MOVL C01664 V=800.0 PL=0
MOVL C01665 V=800.0 PL=0
MOVL C01666 V=800.0 PL=0
MOVL C01667 V=800.0 PL=0
MOVL C01668 V=800.0 PL=0
MOVL C01669 V=800.0 PL=0
MOVL C01670 V=800.0 PL=0
MOVL C01671 V=800.0 PL=0
MOVL C01672 V=800.0 PL=0
MOVL C01673 V=800.0 PL=0
MOVL C01674 V=800.0 PL=0
MOVL C01675 V=800.0 PL=0
MOVL C01676 V=800.0 PL=0
MOVL C01677 V=800.0 PL=0
MOVL C01678 V=800.0 PL=0
MOVL C01679 V=800.0 PL=0
MOVL C01680 V=800.0 PL=0
MOVL C01681 V=800.0 PL=0
MOVL C01682 V=800.0 PL=0
MOVL C01683 V=800.0 PL=0
MOVL C01684 V=800.0 PL=0
MOVL C01685 V=800.0 PL=0
MOVL C01686 V=800.0 PL=0
MOVL C01687 V=800.0 PL=0
MOVL C01688 V=800.0 PL=0
MOVL C01689 V=800.0 PL=0
MOVL C01690 V=800.0 PL=0
MOVL C01691 V=800.0 PL=0
MOVL C01692 V=800.0 PL=0
MOVL C01693 V=800.0 PL=0
MOVL C01694 V=800.0 PL=0
MOVL C01695 V=800.0 PL=0
MOVL C01696 V=800.0 PL=0
MOVL C01697 V=800.0 PL=0
MOVL C01698 V=800.0 PL=0
MOVL C01699 V=800.0 PL=0
MOVL C01700 V=800.0 PL=0
MOVL C01701 V=800.0 PL=0
MOVL C01702 V=800.0 PL=0
MOVL C01703 V=800.0 PL=0
MOVL C01704 V=800.0 PL=0
MOVL C01705 V=800.0 PL=0
MOVL C01706 V=800.0 PL=0
MOVL C01707 V=800.0 PL=0
MOVL C01708 V=800.0 PL=0
MOVL C01709 V=800.0 PL=0
MOVL C01710 V=800.0 PL=0
MOVL C01711 V=800.0 PL=0
MOVL C01712 V=800.0 PL=0
MOVL C01713 V=800.0 PL=0
MOVL C01714 V=800.0 PL=0
MOVL C01715 V=800.0 PL=0
MOVL C01716 V=800.0 PL=0
MOVL C01717 V=800.0 PL=0
MOVL C01718 V=800.0 PL=0
MOVL C01719 V=800.0 PL=0
MOVL C01720 V=800.0 PL=0
MOVL C01721 V=800.0 PL=0
MOVL C01722 V=800.0 PL=0
MOVL C01723 V=800.0 PL=0
MOVL C01724 V=800.0 PL=0
MOVL C01725 V=800.0 PL=0
MOVL C01726 V=800.0 PL=0
MOVL C01727 V=800.0 PL=0
MOVL C01728 V=800.0 PL=0
MOVL C01729 V=800.0 PL=0
MOVL C01730 V=800.0 PL=0
MOVL C01731 V=800.0 PL=0
MOVL C01732 V=800.0 PL=0
MOVL C01733 V=800.0 PL=0
MOVL C01734 V=800.0 PL=0
MOVL C01735 V=800.0 PL=0
MOVL C01736 V=800.0 PL=0
MOVL C01737 V=800.0 PL=0
MOVL C01738 V=800.0 PL=0
MOVL C01739 V=800.0 PL=0
MOVL C01740 V=800.0 PL=0
MOVL C01741 V=800.0 PL=0
MOVL C01742 V=800.0 PL=0
MOVL C01743 V=800.0 PL=0
MOVL C01744 V=800.0 PL=0
MOVL C01745 V=800.0 PL=0
MOVL C01746 V=800.0 PL=0
MOVL C01747 V=800.0 PL=0
MOVL C01748 V=800.0 PL=0
MOVL C01749 V=800.0 PL=0
MOVL C01750 V=800.0 PL=0
MOVL C01751 V=800.0 PL=0
MOVL C01752 V=800.0 PL=0
MOVL C01753 V=800.0 PL=0
MOVL C01754 V=800.0 PL=0
MOVL C01755 V=800.0 PL=0
MOVL C01756 V=800.0 PL=0
MOVL C01757 V=800.0 PL=0
MOVL C01758 V=800.0 PL=0
MOVL C01759 V=800.0 PL=0
MOVL C01760 V=800.0 PL=0
MOVL C01761 V=800.0 PL=0
MOVL C01762 V=800.0 PL=0
MOVL C01763 V=800.0 PL=0
MOVL C01764 V=800.0 PL=0
MOVL C01765 V=800.0 PL=0
MOVL C01766 V=800.0 PL=0
MOVL C01767 V=800.0 PL=0
MOVL C01768 V=800.0 PL=0
MOVL C01769 V=800.0 PL=0
MOVL C01770 V=800.0 PL=0
MOVL C01771 V=800.0 PL=0
MOVL C01772 V=800.0 PL=0
MOVL C01773 V=800.0 PL=0
MOVL C01774 V=800.0 PL=0
MOVL C01775 V=800.0 PL=0
MOVL C01776 V=800.0 PL=0
MOVL C01777 V=800.0 PL=0
MOVL C01778 V=800.0 PL=0
MOVL C01779 V=800.0 PL=0
MOVL C01780 V=800.0 PL=0
MOVL C01781 V=800.0 PL=0
MOVL C01782 V=800.0 PL=0
MOVL C01783 V=800.0 PL=0
MOVL C01784 V=800.0 PL=0
MOVL C01785 V=800.0 PL=0
MOVL C01786 V=800.0 PL=0
MOVL C01787 V=800.0 PL=0
MOVL C01788 V=800.0 PL=0
MOVL C01789 V=800.0 PL=0
MOVL C01790 V=800.0 PL=0
MOVL C01791 V=800.0 PL=0
MOVL C01792 V=800.0 PL=0
MOVL C01793 V=800.0 PL=0
MOVL C01794 V=800.0 PL=0
MOVL C01795 V=800.0 PL=0
MOVL C01796 V=800.0 PL=0
MOVL C01797 V=800.0 PL=0
MOVL C01798 V=800.0 PL=0
MOVL C01799 V=800.0 PL=0
MOVL C01800 V=800.0 PL=0
MOVL C01801 V=800.0 PL=0
MOVL C01802 V=800.0 PL=0
MOVL C01803 V=800.0 PL=0
MOVL C01804 V=800.0 PL=0
MOVL C01805 V=800.0 PL=0
MOVL C01806 V=800.0 PL=0
MOVL C01807 V=800.0 PL=0
MOVL C01808 V=800.0 PL=0
MOVL C01809 V=800.0 PL=0
MOVL C01810 V=800.0 PL=0
MOVL C01811 V=800.0 PL=0
MOVL C01812 V=800.0 PL=0
MOVL C01813 V=800.0 PL=0
MOVL C01814 V=800.0 PL=0
MOVL C01815 V=800.0 PL=0
MOVL C01816 V=800.0 PL=0
MOVL C01817 V=800.0 PL=0
MOVL C01818 V=800.0 PL=0
MOVL C01819 V=800.0 PL=0
MOVL C01820 V=800.0 PL=0
MOVL C01821 V=800.0 PL=0
MOVL C01822 V=800.0 PL=0
MOVL C01823 V=800.0 PL=0
MOVL C01824 V=800.0 PL=0
MOVL C01825 V=800.0 PL=0
MOVL C01826 V=800.0 PL=0
MOVL C01827 V=800.0 PL=0
MOVL C01828 V=800.0 PL=0
MOVL C01829 V=800.0 PL=0
MOVL C01830 V=800.0 PL=0
MOVL C01831 V=800.0 PL=0
MOVL C01832 V=800.0 PL=0
MOVL C01833 V=800.0 PL=0
MOVL C01834 V=800.0 PL=0
MOVL C01835 V=800.0 PL=0
MOVL C01836 V=800.0 PL=0
MOVL C01837 V=800.0 PL=0
MOVL C01838 V=800.0 PL=0
MOVL C01839 V=800.0 PL=0
MOVL C01840 V=800.0 PL=0
MOVL C01841 V=800.0 PL=0
MOVL C01842 V=800.0 PL=0
MOVL C01843 V=800.0 PL=0
MOVL C01844 V=800.0 PL=0
MOVL C01845 V=800.0 PL=0
MOVL C01846 V=800.0 PL=0
MOVL C01847 V=800.0 PL=0
MOVL C01848 V=800.0 PL=0
MOVL C01849 V=800.0 PL=0
MOVL C01850 V=800.0 PL=0
MOVL C01851 V=800.0 PL=0
MOVL C01852 V=800.0 PL=0
MOVL C01853 V=800.0 PL=0
MOVL C01854 V=800.0 PL=0
MOVL C01855 V=800.0 PL=0
MOVL C01856 V=800.0 PL=0
MOVL C01857 V=800.0 PL=0
MOVL C01858 V=800.0 PL=0
MOVL C01859 V=800.0 PL=0
MOVL C01860 V=800.0 PL=0
MOVL C01861 V=800.0 PL=0
MOVL C01862 V=800.0 PL=0
MOVL C01863 V=800.0 PL=0
MOVL C01864 V=800.0 PL=0
MOVL C01865 V=800.0 PL=0
MOVL C01866 V=800.0 PL=0
MOVL C01867 V=800.0 PL=0
MOVL C01868 V=800.0 PL=0
MOVL C01869 V=800.0 PL=0
MOVL C01870 V=800.0 PL=0
MOVL C01871 V=800.0 PL=0
MOVL C01872 V=800.0 PL=0
MOVL C01873 V=800.0 PL=0
MOVL C01874 V=800.0 PL=0
MOVL C01875 V=800.0 PL=0
MOVL C01876 V=800.0 PL=0
MOVL C01877 V=800.0 PL=0
MOVL C01878 V=800.0 PL=0
MOVL C01879 V=800.0 PL=0
MOVL C01880 V=800.0 PL=0
MOVL C01881 V=800.0 PL=0
MOVL C01882 V=800.0 PL=0
MOVL C01883 V=800.0 PL=0
MOVL C01884 V=800.0 PL=0
MOVL C01885 V=800.0 PL=0
MOVL C01886 V=800.0 PL=0
MOVL C01887 V=800.0 PL=0
MOVL C01888 V=800.0 PL=0
MOVL C01889 V=800.0 PL=0
MOVL C01890 V=800.0 PL=0
MOVL C01891 V=800.0 PL=0
MOVL C01892 V=800.0 PL=0
MOVL C01893 V=800.0 PL=0
MOVL C01894 V=800.0 PL=0
MOVL C01895 V=800.0 PL=0
MOVL C01896 V=800.0 PL=0
MOVL C01897 V=800.0 PL=0
MOVL C01898 V=800.0 PL=0
MOVL C01899 V=800.0 PL=0
MOVL C01900 V=800.0 PL=0
MOVL C01901 V=800.0 PL=0
MOVL C01902 V=800.0 PL=0
MOVL C01903 V=800.0 PL=0
MOVL C01904 V=800.0 PL=0
MOVL C01905 V=800.0 PL=0
MOVL C01906 V=800.0 PL=0
MOVL C01907 V=800.0 PL=0
MOVL C01908 V=800.0 PL=0
MOVL C01909 V=800.0 PL=0
MOVL C01910 V=800.0 PL=0
MOVL C01911 V=800.0 PL=0
MOVL C01912 V=800.0 PL=0
MOVL C01913 V=800.0 PL=0
MOVL C01914 V=800.0 PL=0
MOVL C01915 V=800.0 PL=0
MOVL C01916 V=800.0 PL=0
MOVL C01917 V=800.0 PL=0
MOVL C01918 V=800.0 PL=0
MOVL C01919 V=800.0 PL=0
MOVL C01920 V=800.0 PL=0
MOVL C01921 V=800.0 PL=0
MOVL C01922 V=800.0 PL=0
MOVL C01923 V=800.0 PL=0
MOVL C01924 V=800.0 PL=0
MOVL C01925 V=800.0 PL=0
MOVL C01926 V=800.0 PL=0
MOVL C01927 V=800.0 PL=0
MOVL C01928 V=800.0 PL=0
MOVL C01929 V=800.0 PL=0
MOVL C01930 V=800.0 PL=0
MOVL C01931 V=800.0 PL=0
MOVL C01932 V=800.0 PL=0
MOVL C01933 V=800.0 PL=0
MOVL C01934 V=800.0 PL=0
MOVL C01935 V=800.0 PL=0
MOVL C01936 V=800.0 PL=0
MOVL C01937 V=800.0 PL=0
MOVL C01938 V=800.0 PL=0
MOVL C01939 V=800.0 PL=0
MOVL C01940 V=800.0 PL=0
MOVL C01941 V=800.0 PL=0
MOVL C01942 V=800.0 PL=0
MOVL C01943 V=800.0 PL=0
MOVL C01944 V=800.0 PL=0
MOVL C01945 V=800.0 PL=0
MOVL C01946 V=800.0 PL=0
MOVL C01947 V=800.0 PL=0
MOVL C01948 V=800.0 PL=0
MOVL C01949 V=800.0 PL=0
MOVL C01950 V=800.0 PL=0
MOVL C01951 V=800.0 PL=0
MOVL C01952 V=800.0 PL=0
MOVL C01953 V=800.0 PL=0
MOVL C01954 V=800.0 PL=0
MOVL C01955 V=800.0 PL=0
MOVL C01956 V=800.0 PL=0
MOVL C01957 V=800.0 PL=0
MOVL C01958 V=800.0 PL=0
MOVL C01959 V=800.0 PL=0
MOVL C01960 V=800.0 PL=0
MOVL C01961 V=800.0 PL=0
MOVL C01962 V=800.0 PL=0
MOVL C01963 V=800.0 PL=0
MOVL C01964 V=800.0 PL=0
MOVL C01965 V=800.0 PL=0
MOVL C01966 V=800.0 PL=0
MOVL C01967 V=800.0 PL=0
MOVL C01968 V=800.0 PL=0
MOVL C01969 V=800.0 PL=0
MOVL C01970 V=800.0 PL=0
MOVL C01971 V=800.0 PL=0
MOVL C01972 V=800.0 PL=0
MOVL C01973 V=800.0 PL=0
MOVL C01974 V=800.0 PL=0
MOVL C01975 V=800.0 PL=0
MOVL C01976 V=800.0 PL=0
MOVL C01977 V=800.0 PL=0
MOVL C01978 V=800.0 PL=0
MOVL C01979 V=800.0 PL=0
MOVL C01980 V=800.0 PL=0
MOVL C01981 V=800.0 PL=0
MOVL C01982 V=800.0 PL=0
MOVL C01983 V=800.0 PL=0
MOVL C01984 V=800.0 PL=0
MOVL C01985 V=800.0 PL=0
MOVL C01986 V=800.0 PL=0
MOVL C01987 V=800.0 PL=0
MOVL C01988 V=800.0 PL=0
MOVL C01989 V=800.0 PL=0
MOVL C01990 V=800.0 PL=0
MOVL C01991 V=800.0 PL=0
MOVL C01992 V=800.0 PL=0
MOVL C01993 V=800.0 PL=0
MOVL C01994 V=800.0 PL=0
MOVL C01995 V=800.0 PL=0
MOVL C01996 V=800.0 PL=0
MOVL C01997 V=800.0 PL=0
MOVL C01998 V=800.0 PL=0
MOVL C01999 V=800.0 PL=0
MOVL C02000 V=800.0 PL=0
MOVL C02001 V=800.0 PL=0
MOVL C02002 V=800.0 PL=0
MOVL C02003 V=800.0 PL=0
MOVL C02004 V=800.0 PL=0
